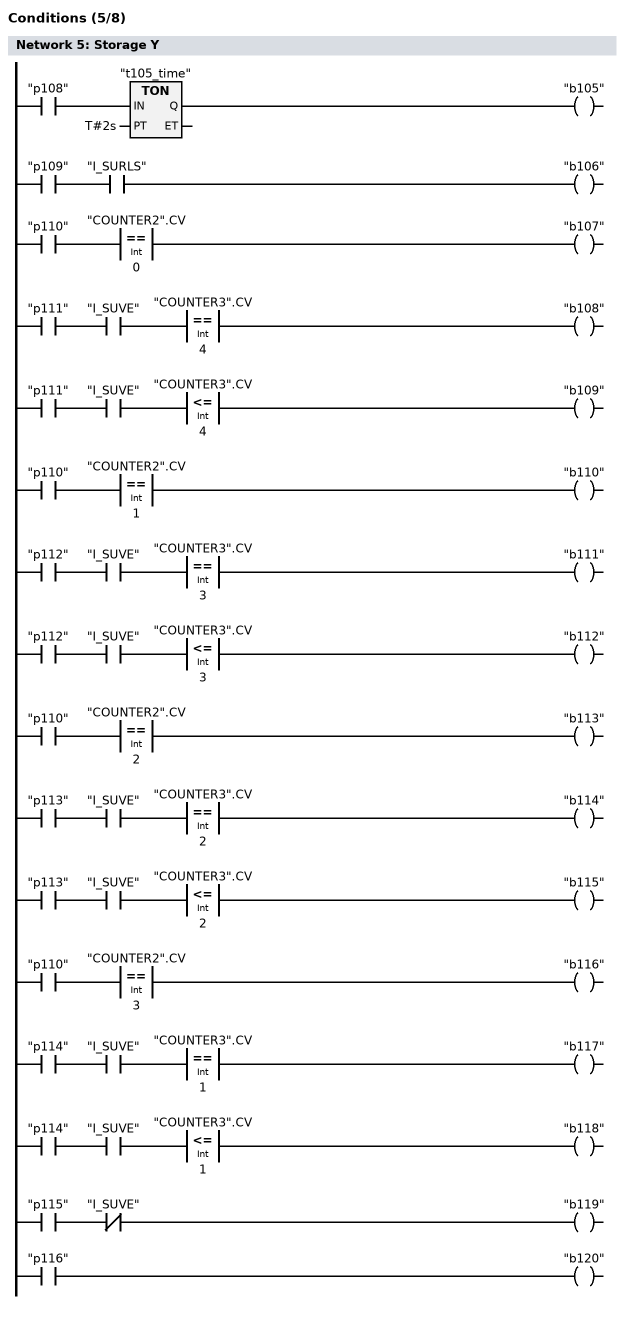
   "t105_time".TON(IN := "p108", PT := T#2s);
   "b105" := "t105_time".Q;
   "b106" := "p109" AND "I_SURLS";
   "b107" := "p110" AND ("COUNTER2".CV = 0);
   "b108" := "p111" AND "I_SUVE" AND ("COUNTER3".CV = 4);
   "b109" := "p111" AND "I_SUVE" AND ("COUNTER3".CV <= 4);
   "b110" := "p110" AND ("COUNTER2".CV = 1);
   "b111" := "p112" AND "I_SUVE" AND ("COUNTER3".CV = 3);
   "b112" := "p112" AND "I_SUVE" AND ("COUNTER3".CV <= 3);
   "b113" := "p110" AND ("COUNTER2".CV = 2);
   "b114" := "p113" AND "I_SUVE" AND ("COUNTER3".CV = 2);
   "b115" := "p113" AND "I_SUVE" AND ("COUNTER3".CV <= 2);
   "b116" := "p110" AND ("COUNTER2".CV = 3);
   "b117" := "p114" AND "I_SUVE" AND ("COUNTER3".CV = 1);
   "b118" := "p114" AND "I_SUVE" AND ("COUNTER3".CV <= 1);
   "b119" := "p115" AND NOT "I_SUVE";
   "b120" := "p116";
END_REGION

REGION Network 6: Storage X
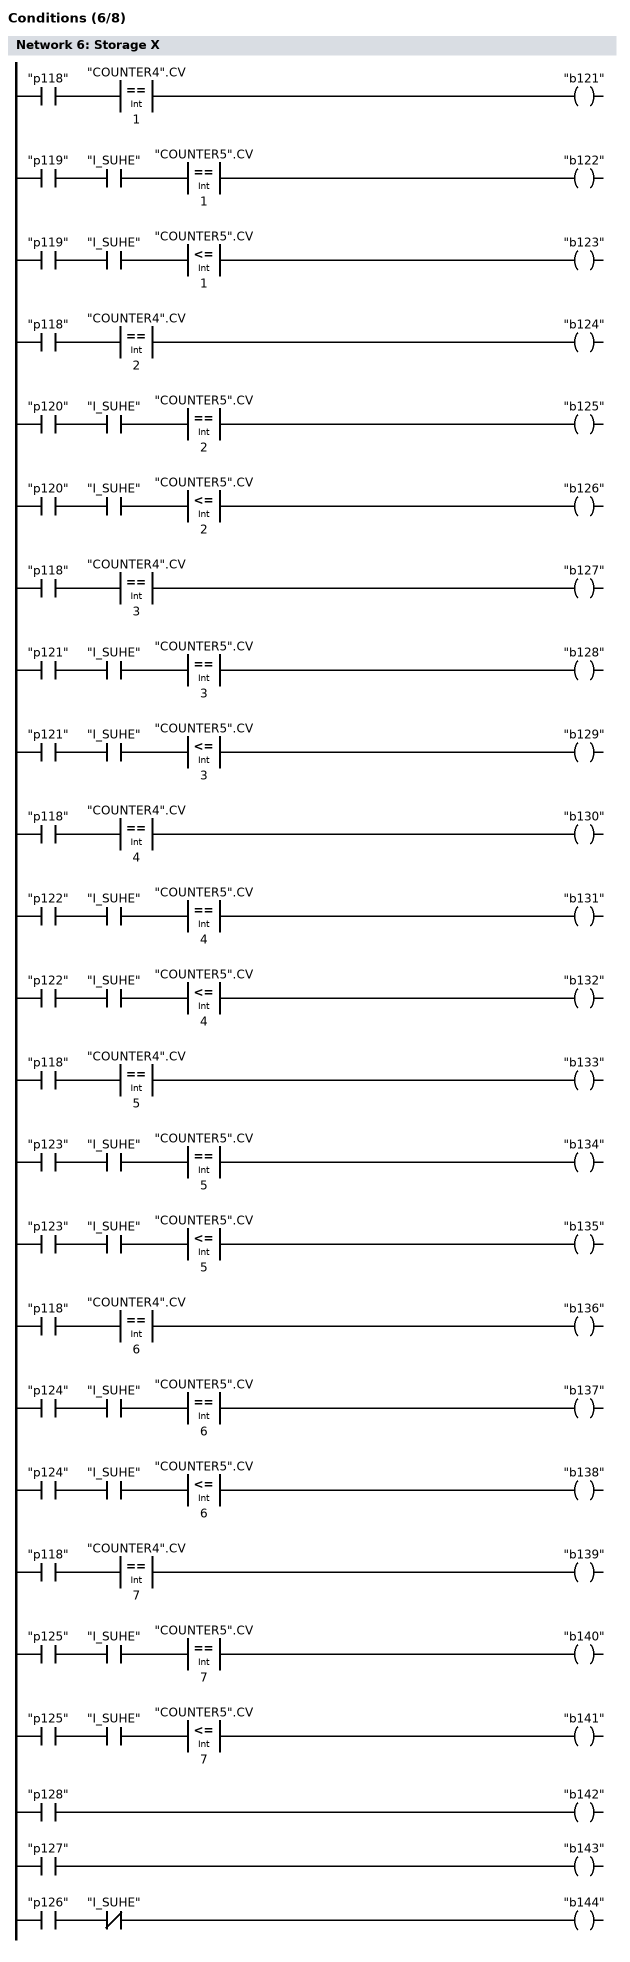
   RUNG wire#powerrail
      Contact( "p118" )
      { S7_Templates := "SrcType := Int" } EQ_Contact(in1 := "COUNTER4".CV, in2 := 1)
      Coil( "b121" )
   END_RUNG
   RUNG wire#powerrail
      Contact( "p119" )
      Contact( "I_SUHE" )
      { S7_Templates := "SrcType := Int" } EQ_Contact(in1 := "COUNTER5".CV, in2 := 1)
      Coil( "b122" )
   END_RUNG
   RUNG wire#powerrail
      Contact( "p119" )
      Contact( "I_SUHE" )
      { S7_Templates := "SrcType := Int" } LE_Contact(in1 := "COUNTER5".CV, in2 := 1)
      Coil( "b123" )
   END_RUNG
   RUNG wire#powerrail
      Contact( "p118" )
      { S7_Templates := "SrcType := Int" } EQ_Contact(in1 := "COUNTER4".CV, in2 := 2)
      Coil( "b124" )
   END_RUNG
   RUNG wire#powerrail
      Contact( "p120" )
      Contact( "I_SUHE" )
      { S7_Templates := "SrcType := Int" } EQ_Contact(in1 := "COUNTER5".CV, in2 := 2)
      Coil( "b125" )
   END_RUNG
   RUNG wire#powerrail
      Contact( "p120" )
      Contact( "I_SUHE" )
      { S7_Templates := "SrcType := Int" } LE_Contact(in1 := "COUNTER5".CV, in2 := 2)
      Coil( "b126" )
   END_RUNG
   RUNG wire#powerrail
      Contact( "p118" )
      { S7_Templates := "SrcType := Int" } EQ_Contact(in1 := "COUNTER4".CV, in2 := 3)
      Coil( "b127" )
   END_RUNG
   RUNG wire#powerrail
      Contact( "p121" )
      Contact( "I_SUHE" )
      { S7_Templates := "SrcType := Int" } EQ_Contact(in1 := "COUNTER5".CV, in2 := 3)
      Coil( "b128" )
   END_RUNG
   RUNG wire#powerrail
      Contact( "p121" )
      Contact( "I_SUHE" )
      { S7_Templates := "SrcType := Int" } LE_Contact(in1 := "COUNTER5".CV, in2 := 3)
      Coil( "b129" )
   END_RUNG
   RUNG wire#powerrail
      Contact( "p118" )
      { S7_Templates := "SrcType := Int" } EQ_Contact(in1 := "COUNTER4".CV, in2 := 4)
      Coil( "b130" )
   END_RUNG
   RUNG wire#powerrail
      Contact( "p122" )
      Contact( "I_SUHE" )
      { S7_Templates := "SrcType := Int" } EQ_Contact(in1 := "COUNTER5".CV, in2 := 4)
      Coil( "b131" )
   END_RUNG
   RUNG wire#powerrail
      Contact( "p122" )
      Contact( "I_SUHE" )
      { S7_Templates := "SrcType := Int" } LE_Contact(in1 := "COUNTER5".CV, in2 := 4)
      Coil( "b132" )
   END_RUNG
   RUNG wire#powerrail
      Contact( "p118" )
      { S7_Templates := "SrcType := Int" } EQ_Contact(in1 := "COUNTER4".CV, in2 := 5)
      Coil( "b133" )
   END_RUNG
   RUNG wire#powerrail
      Contact( "p123" )
      Contact( "I_SUHE" )
      { S7_Templates := "SrcType := Int" } EQ_Contact(in1 := "COUNTER5".CV, in2 := 5)
      Coil( "b134" )
   END_RUNG
   RUNG wire#powerrail
      Contact( "p123" )
      Contact( "I_SUHE" )
      { S7_Templates := "SrcType := Int" } LE_Contact(in1 := "COUNTER5".CV, in2 := 5)
      Coil( "b135" )
   END_RUNG
   RUNG wire#powerrail
      Contact( "p118" )
      { S7_Templates := "SrcType := Int" } EQ_Contact(in1 := "COUNTER4".CV, in2 := 6)
      Coil( "b136" )
   END_RUNG
   RUNG wire#powerrail
      Contact( "p124" )
      Contact( "I_SUHE" )
      { S7_Templates := "SrcType := Int" } EQ_Contact(in1 := "COUNTER5".CV, in2 := 6)
      Coil( "b137" )
   END_RUNG
   RUNG wire#powerrail
      Contact( "p124" )
      Contact( "I_SUHE" )
      { S7_Templates := "SrcType := Int" } LE_Contact(in1 := "COUNTER5".CV, in2 := 6)
      Coil( "b138" )
   END_RUNG
   RUNG wire#powerrail
      Contact( "p118" )
      { S7_Templates := "SrcType := Int" } EQ_Contact(in1 := "COUNTER4".CV, in2 := 7)
      Coil( "b139" )
   END_RUNG
   RUNG wire#powerrail
      Contact( "p125" )
      Contact( "I_SUHE" )
      { S7_Templates := "SrcType := Int" } EQ_Contact(in1 := "COUNTER5".CV, in2 := 7)
      Coil( "b140" )
   END_RUNG
   RUNG wire#powerrail
      Contact( "p125" )
      Contact( "I_SUHE" )
      { S7_Templates := "SrcType := Int" } LE_Contact(in1 := "COUNTER5".CV, in2 := 7)
      Coil( "b141" )
   END_RUNG
   RUNG wire#powerrail
      Contact( "p128" )
      Coil( "b142" )
   END_RUNG
   RUNG wire#powerrail
      Contact( "p127" )
      Coil( "b143" )
   END_RUNG
   RUNG wire#powerrail
      Contact( "p126" )
      I_Contact( "I_SUHE" )
      Coil( "b144" )
   END_RUNG
   // the same network as SCL:
   "b121" := "p118" AND ("COUNTER4".CV = 1);
   "b122" := "p119" AND "I_SUHE" AND ("COUNTER5".CV = 1);
   "b123" := "p119" AND "I_SUHE" AND ("COUNTER5".CV <= 1);
   "b124" := "p118" AND ("COUNTER4".CV = 2);
   "b125" := "p120" AND "I_SUHE" AND ("COUNTER5".CV = 2);
   "b126" := "p120" AND "I_SUHE" AND ("COUNTER5".CV <= 2);
   "b127" := "p118" AND ("COUNTER4".CV = 3);
   "b128" := "p121" AND "I_SUHE" AND ("COUNTER5".CV = 3);
   "b129" := "p121" AND "I_SUHE" AND ("COUNTER5".CV <= 3);
   "b130" := "p118" AND ("COUNTER4".CV = 4);
   "b131" := "p122" AND "I_SUHE" AND ("COUNTER5".CV = 4);
   "b132" := "p122" AND "I_SUHE" AND ("COUNTER5".CV <= 4);
   "b133" := "p118" AND ("COUNTER4".CV = 5);
   "b134" := "p123" AND "I_SUHE" AND ("COUNTER5".CV = 5);
   "b135" := "p123" AND "I_SUHE" AND ("COUNTER5".CV <= 5);
   "b136" := "p118" AND ("COUNTER4".CV = 6);
   "b137" := "p124" AND "I_SUHE" AND ("COUNTER5".CV = 6);
   "b138" := "p124" AND "I_SUHE" AND ("COUNTER5".CV <= 6);
   "b139" := "p118" AND ("COUNTER4".CV = 7);
   "b140" := "p125" AND "I_SUHE" AND ("COUNTER5".CV = 7);
   "b141" := "p125" AND "I_SUHE" AND ("COUNTER5".CV <= 7);
   "b142" := "p128";
   "b143" := "p127";
   "b144" := "p126" AND NOT "I_SUHE";
END_REGION

REGION Network 7: Storage piece
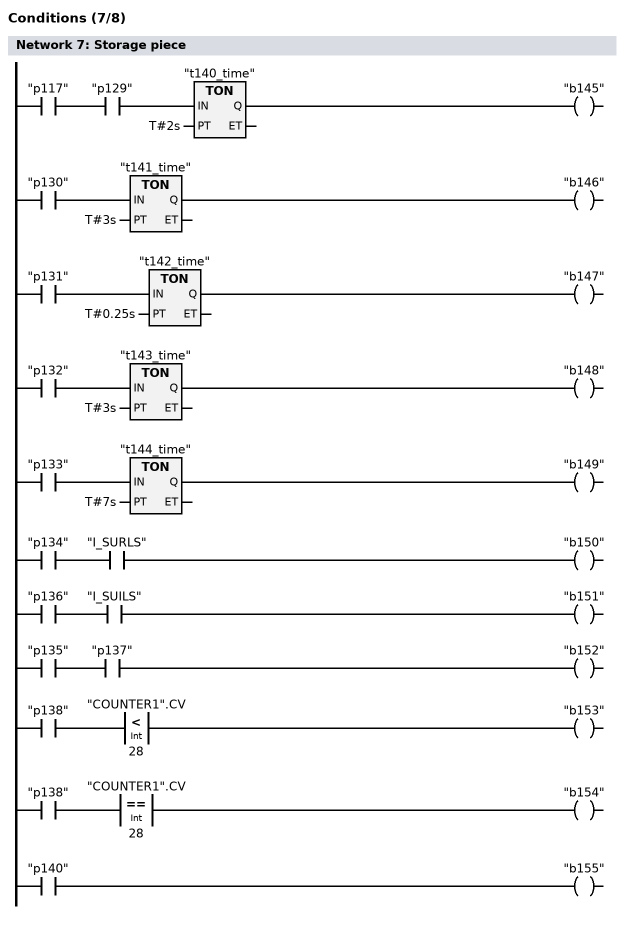
   "t140_time".TON(IN := "p117" AND "p129", PT := T#2s);
   "b145" := "t140_time".Q;
   "t141_time".TON(IN := "p130", PT := T#3s);
   "b146" := "t141_time".Q;
   "t142_time".TON(IN := "p131", PT := T#0.25s);
   "b147" := "t142_time".Q;
   "t143_time".TON(IN := "p132", PT := T#3s);
   "b148" := "t143_time".Q;
   "t144_time".TON(IN := "p133", PT := T#7s);
   "b149" := "t144_time".Q;
   "b150" := "p134" AND "I_SURLS";
   "b151" := "p136" AND "I_SUILS";
   "b152" := "p135" AND "p137";
   "b153" := "p138" AND ("COUNTER1".CV < 28);
   "b154" := "p138" AND ("COUNTER1".CV = 28);
   "b155" := "p140";
END_REGION

REGION Network 8: Arm Stop
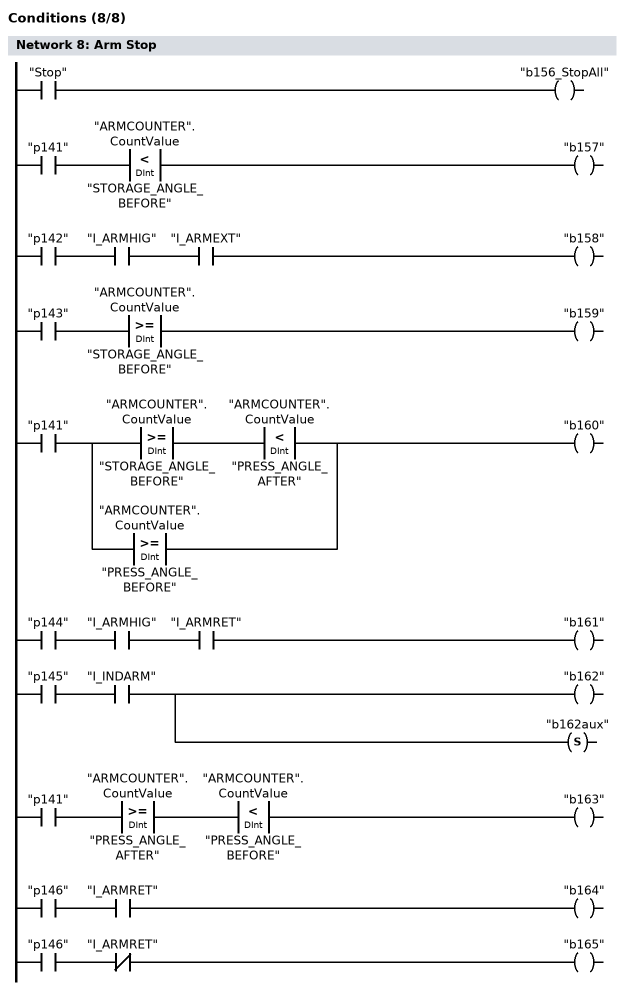
   RUNG wire#powerrail
      Contact( "Stop" )
      Coil( "b156_StopAll" )
   END_RUNG
   RUNG wire#powerrail
      Contact( "p141" )
      { S7_Templates := "SrcType := DInt" } LT_Contact(in1 := "ARMCOUNTER".CountValue, in2 := "STORAGE_ANGLE_BEFORE")
      Coil( "b157" )
   END_RUNG
   RUNG wire#powerrail
      Contact( "p142" )
      Contact( "I_ARMHIG" )
      Contact( "I_ARMEXT" )
      Coil( "b158" )
   END_RUNG
   RUNG wire#powerrail
      Contact( "p143" )
      { S7_Templates := "SrcType := DInt" } GE_Contact(in1 := "ARMCOUNTER".CountValue, in2 := "STORAGE_ANGLE_BEFORE")
      Coil( "b159" )
   END_RUNG
   RUNG wire#powerrail
      Contact( "p141" )
      wire#w1
      { S7_Templates := "SrcType := DInt" } GE_Contact(in1 := "ARMCOUNTER".CountValue, in2 := "STORAGE_ANGLE_BEFORE")
      { S7_Templates := "SrcType := DInt" } LT_Contact(in1 := "ARMCOUNTER".CountValue, in2 := "PRESS_ANGLE_AFTER")
      wire#w2
      Coil( "b160" )
   END_RUNG
   RUNG wire#w1
      { S7_Templates := "SrcType := DInt" } GE_Contact(in1 := "ARMCOUNTER".CountValue, in2 := "PRESS_ANGLE_BEFORE")
   END_RUNG wire#w2
   RUNG wire#powerrail
      Contact( "p144" )
      Contact( "I_ARMHIG" )
      Contact( "I_ARMRET" )
      Coil( "b161" )
   END_RUNG
   RUNG wire#powerrail
      Contact( "p145" )
      Contact( "I_INDARM" )
      wire#w3
      Coil( "b162" )
   END_RUNG
   RUNG wire#w3
      S_Coil( "b162aux" )
   END_RUNG
   RUNG wire#powerrail
      Contact( "p141" )
      { S7_Templates := "SrcType := DInt" } GE_Contact(in1 := "ARMCOUNTER".CountValue, in2 := "PRESS_ANGLE_AFTER")
      { S7_Templates := "SrcType := DInt" } LT_Contact(in1 := "ARMCOUNTER".CountValue, in2 := "PRESS_ANGLE_BEFORE")
      Coil( "b163" )
   END_RUNG
   RUNG wire#powerrail
      Contact( "p146" )
      Contact( "I_ARMRET" )
      Coil( "b164" )
   END_RUNG
   RUNG wire#powerrail
      Contact( "p146" )
      I_Contact( "I_ARMRET" )
      Coil( "b165" )
   END_RUNG
   // the same network as SCL:
   "b156_StopAll" := "Stop";
   "b157" := "p141" AND ("ARMCOUNTER".CountValue < "STORAGE_ANGLE_BEFORE");
   "b158" := "p142" AND "I_ARMHIG" AND "I_ARMEXT";
   "b159" := "p143" AND ("ARMCOUNTER".CountValue >= "STORAGE_ANGLE_BEFORE");
   "b160" := "p141" AND ((("ARMCOUNTER".CountValue >= "STORAGE_ANGLE_BEFORE") AND ("ARMCOUNTER".CountValue < "PRESS_ANGLE_AFTER")) OR ("ARMCOUNTER".CountValue >= "PRESS_ANGLE_BEFORE"));
   "b161" := "p144" AND "I_ARMHIG" AND "I_ARMRET";
   "b162" := "p145" AND "I_INDARM";
   IF "b162" THEN "b162aux" := TRUE; END_IF;
   "b163" := "p141" AND ("ARMCOUNTER".CountValue >= "PRESS_ANGLE_AFTER") AND ("ARMCOUNTER".CountValue < "PRESS_ANGLE_BEFORE");
   "b164" := "p146" AND "I_ARMRET";
   "b165" := "p146" AND NOT "I_ARMRET";
END_REGION
END_FUNCTION

FUNCTION "Dynamics" : Void   // FC3, LAD
{ S7_Optimized_Access := 'TRUE' }
VERSION : 0.1
BEGIN

REGION Network 1: initialization
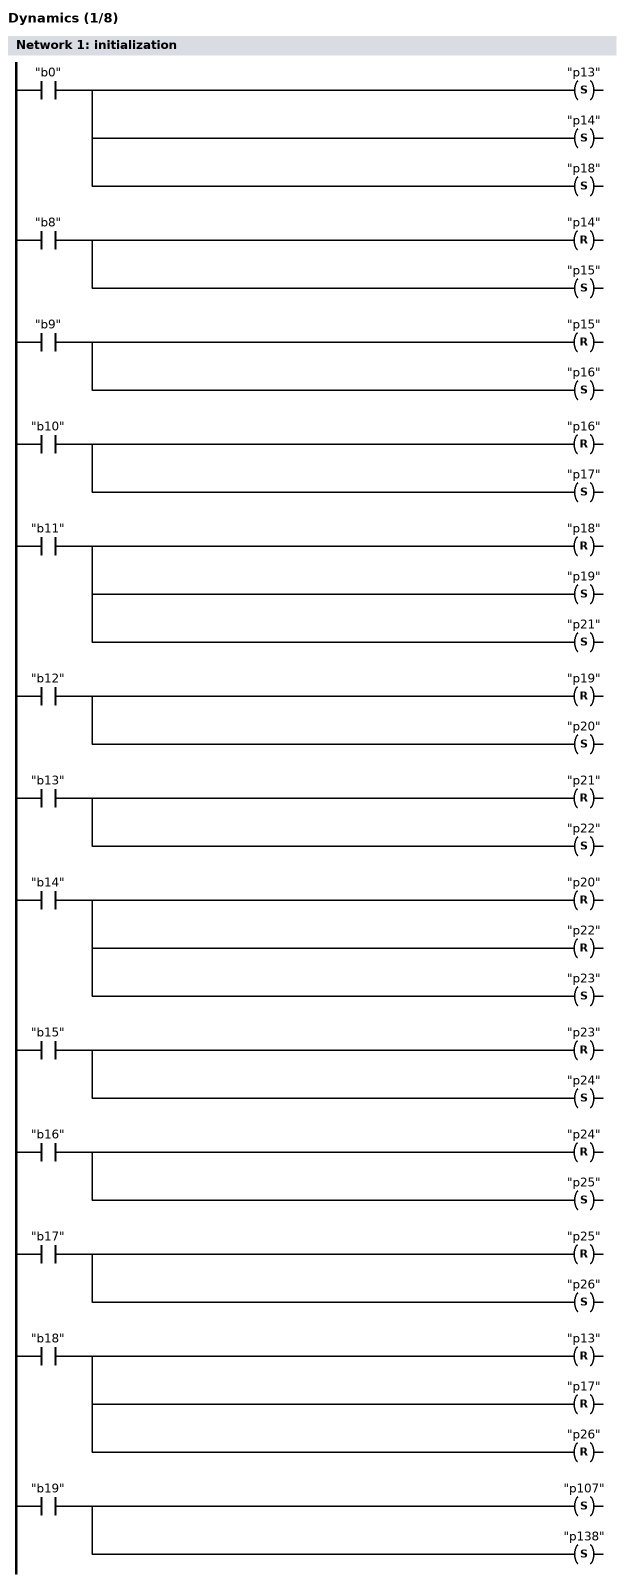
   RUNG wire#powerrail
      Contact( "b0" )
      wire#w1
      S_Coil( "p13" )
   END_RUNG
   RUNG wire#w1
      S_Coil( "p14" )
   END_RUNG
   RUNG wire#w1
      S_Coil( "p18" )
   END_RUNG
   RUNG wire#powerrail
      Contact( "b8" )
      wire#w2
      R_Coil( "p14" )
   END_RUNG
   RUNG wire#w2
      S_Coil( "p15" )
   END_RUNG
   RUNG wire#powerrail
      Contact( "b9" )
      wire#w3
      R_Coil( "p15" )
   END_RUNG
   RUNG wire#w3
      S_Coil( "p16" )
   END_RUNG
   RUNG wire#powerrail
      Contact( "b10" )
      wire#w4
      R_Coil( "p16" )
   END_RUNG
   RUNG wire#w4
      S_Coil( "p17" )
   END_RUNG
   RUNG wire#powerrail
      Contact( "b11" )
      wire#w5
      R_Coil( "p18" )
   END_RUNG
   RUNG wire#w5
      S_Coil( "p19" )
   END_RUNG
   RUNG wire#w5
      S_Coil( "p21" )
   END_RUNG
   RUNG wire#powerrail
      Contact( "b12" )
      wire#w6
      R_Coil( "p19" )
   END_RUNG
   RUNG wire#w6
      S_Coil( "p20" )
   END_RUNG
   RUNG wire#powerrail
      Contact( "b13" )
      wire#w7
      R_Coil( "p21" )
   END_RUNG
   RUNG wire#w7
      S_Coil( "p22" )
   END_RUNG
   RUNG wire#powerrail
      Contact( "b14" )
      wire#w8
      R_Coil( "p20" )
   END_RUNG
   RUNG wire#w8
      R_Coil( "p22" )
   END_RUNG
   RUNG wire#w8
      S_Coil( "p23" )
   END_RUNG
   RUNG wire#powerrail
      Contact( "b15" )
      wire#w9
      R_Coil( "p23" )
   END_RUNG
   RUNG wire#w9
      S_Coil( "p24" )
   END_RUNG
   RUNG wire#powerrail
      Contact( "b16" )
      wire#w10
      R_Coil( "p24" )
   END_RUNG
   RUNG wire#w10
      S_Coil( "p25" )
   END_RUNG
   RUNG wire#powerrail
      Contact( "b17" )
      wire#w11
      R_Coil( "p25" )
   END_RUNG
   RUNG wire#w11
      S_Coil( "p26" )
   END_RUNG
   RUNG wire#powerrail
      Contact( "b18" )
      wire#w12
      R_Coil( "p13" )
   END_RUNG
   RUNG wire#w12
      R_Coil( "p17" )
   END_RUNG
   RUNG wire#w12
      R_Coil( "p26" )
   END_RUNG
   RUNG wire#powerrail
      Contact( "b19" )
      wire#w13
      S_Coil( "p107" )
   END_RUNG
   RUNG wire#w13
      S_Coil( "p138" )
   END_RUNG
   // the same network as SCL:
   IF "b0" THEN
       "p13" := TRUE;
       "p14" := TRUE;
       "p18" := TRUE;
   END_IF;
   IF "b8" THEN
       "p14" := FALSE;
       "p15" := TRUE;
   END_IF;
   IF "b9" THEN
       "p15" := FALSE;
       "p16" := TRUE;
   END_IF;
   IF "b10" THEN
       "p16" := FALSE;
       "p17" := TRUE;
   END_IF;
   IF "b11" THEN
       "p18" := FALSE;
       "p19" := TRUE;
       "p21" := TRUE;
   END_IF;
   IF "b12" THEN
       "p19" := FALSE;
       "p20" := TRUE;
   END_IF;
   IF "b13" THEN
       "p21" := FALSE;
       "p22" := TRUE;
   END_IF;
   IF "b14" THEN
       "p20" := FALSE;
       "p22" := FALSE;
       "p23" := TRUE;
   END_IF;
   IF "b15" THEN
       "p23" := FALSE;
       "p24" := TRUE;
   END_IF;
   IF "b16" THEN
       "p24" := FALSE;
       "p25" := TRUE;
   END_IF;
   IF "b17" THEN
       "p25" := FALSE;
       "p26" := TRUE;
   END_IF;
   IF "b18" THEN
       "p13" := FALSE;
       "p17" := FALSE;
       "p26" := FALSE;
   END_IF;
   IF "b19" THEN
       "p107" := TRUE;
       "p138" := TRUE;
   END_IF;
END_REGION

REGION Network 3: Arm Belt to Press
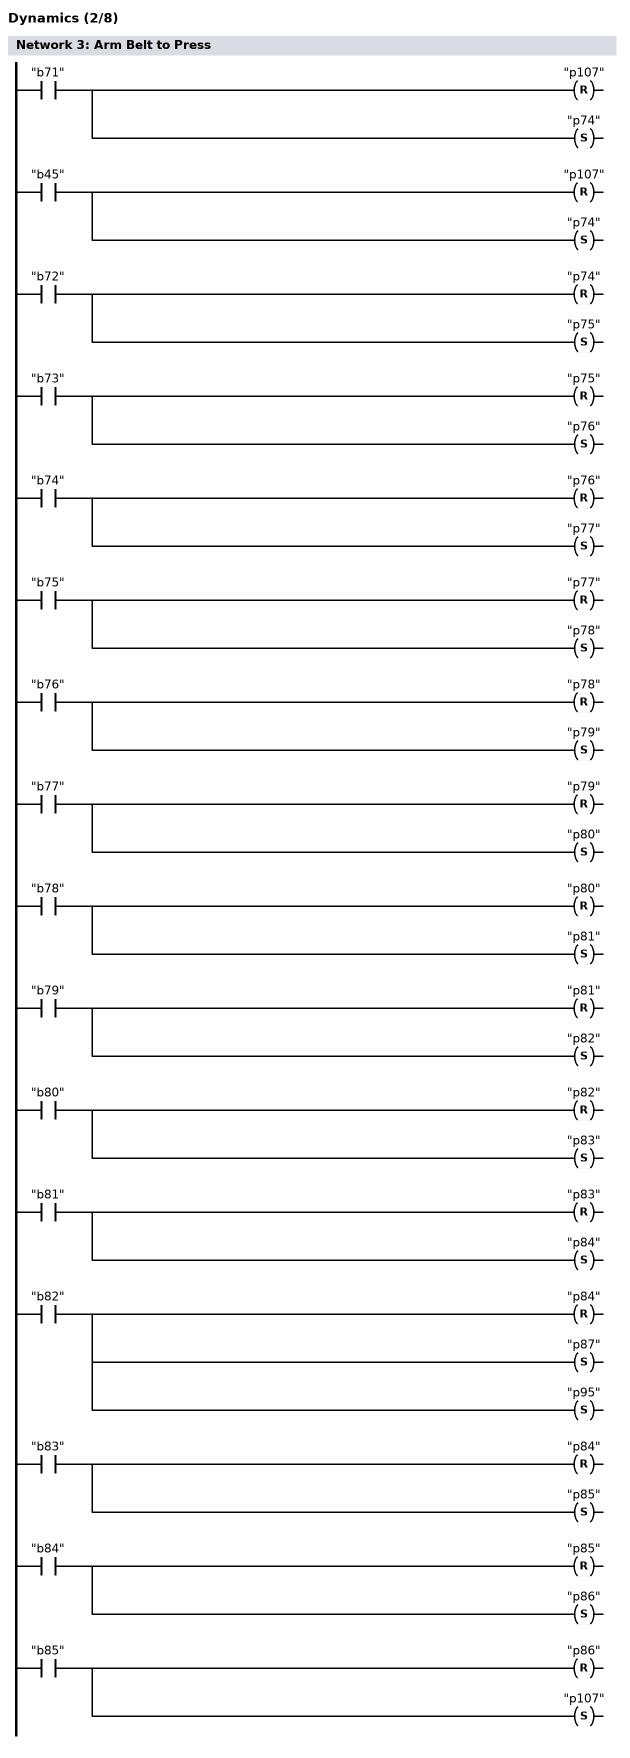
   RUNG wire#powerrail
      Contact( "b71" )
      wire#w1
      R_Coil( "p107" )
   END_RUNG
   RUNG wire#w1
      S_Coil( "p74" )
   END_RUNG
   RUNG wire#powerrail
      Contact( "b45" )
      wire#w2
      R_Coil( "p107" )
   END_RUNG
   RUNG wire#w2
      S_Coil( "p74" )
   END_RUNG
   RUNG wire#powerrail
      Contact( "b72" )
      wire#w3
      R_Coil( "p74" )
   END_RUNG
   RUNG wire#w3
      S_Coil( "p75" )
   END_RUNG
   RUNG wire#powerrail
      Contact( "b73" )
      wire#w4
      R_Coil( "p75" )
   END_RUNG
   RUNG wire#w4
      S_Coil( "p76" )
   END_RUNG
   RUNG wire#powerrail
      Contact( "b74" )
      wire#w5
      R_Coil( "p76" )
   END_RUNG
   RUNG wire#w5
      S_Coil( "p77" )
   END_RUNG
   RUNG wire#powerrail
      Contact( "b75" )
      wire#w6
      R_Coil( "p77" )
   END_RUNG
   RUNG wire#w6
      S_Coil( "p78" )
   END_RUNG
   RUNG wire#powerrail
      Contact( "b76" )
      wire#w7
      R_Coil( "p78" )
   END_RUNG
   RUNG wire#w7
      S_Coil( "p79" )
   END_RUNG
   RUNG wire#powerrail
      Contact( "b77" )
      wire#w8
      R_Coil( "p79" )
   END_RUNG
   RUNG wire#w8
      S_Coil( "p80" )
   END_RUNG
   RUNG wire#powerrail
      Contact( "b78" )
      wire#w9
      R_Coil( "p80" )
   END_RUNG
   RUNG wire#w9
      S_Coil( "p81" )
   END_RUNG
   RUNG wire#powerrail
      Contact( "b79" )
      wire#w10
      R_Coil( "p81" )
   END_RUNG
   RUNG wire#w10
      S_Coil( "p82" )
   END_RUNG
   RUNG wire#powerrail
      Contact( "b80" )
      wire#w11
      R_Coil( "p82" )
   END_RUNG
   RUNG wire#w11
      S_Coil( "p83" )
   END_RUNG
   RUNG wire#powerrail
      Contact( "b81" )
      wire#w12
      R_Coil( "p83" )
   END_RUNG
   RUNG wire#w12
      S_Coil( "p84" )
   END_RUNG
   RUNG wire#powerrail
      Contact( "b82" )
      wire#w13
      R_Coil( "p84" )
   END_RUNG
   RUNG wire#w13
      S_Coil( "p87" )
   END_RUNG
   RUNG wire#w13
      S_Coil( "p95" )
   END_RUNG
   RUNG wire#powerrail
      Contact( "b83" )
      wire#w14
      R_Coil( "p84" )
   END_RUNG
   RUNG wire#w14
      S_Coil( "p85" )
   END_RUNG
   RUNG wire#powerrail
      Contact( "b84" )
      wire#w15
      R_Coil( "p85" )
   END_RUNG
   RUNG wire#w15
      S_Coil( "p86" )
   END_RUNG
   RUNG wire#powerrail
      Contact( "b85" )
      wire#w16
      R_Coil( "p86" )
   END_RUNG
   RUNG wire#w16
      S_Coil( "p107" )
   END_RUNG
   // the same network as SCL:
   IF "b71" THEN
       "p107" := FALSE;
       "p74" := TRUE;
   END_IF;
   IF "b45" THEN
       "p107" := FALSE;
       "p74" := TRUE;
   END_IF;
   IF "b72" THEN
       "p74" := FALSE;
       "p75" := TRUE;
   END_IF;
   IF "b73" THEN
       "p75" := FALSE;
       "p76" := TRUE;
   END_IF;
   IF "b74" THEN
       "p76" := FALSE;
       "p77" := TRUE;
   END_IF;
   IF "b75" THEN
       "p77" := FALSE;
       "p78" := TRUE;
   END_IF;
   IF "b76" THEN
       "p78" := FALSE;
       "p79" := TRUE;
   END_IF;
   IF "b77" THEN
       "p79" := FALSE;
       "p80" := TRUE;
   END_IF;
   IF "b78" THEN
       "p80" := FALSE;
       "p81" := TRUE;
   END_IF;
   IF "b79" THEN
       "p81" := FALSE;
       "p82" := TRUE;
   END_IF;
   IF "b80" THEN
       "p82" := FALSE;
       "p83" := TRUE;
   END_IF;
   IF "b81" THEN
       "p83" := FALSE;
       "p84" := TRUE;
   END_IF;
   IF "b82" THEN
       "p84" := FALSE;
       "p87" := TRUE;
       "p95" := TRUE;
   END_IF;
   IF "b83" THEN
       "p84" := FALSE;
       "p85" := TRUE;
   END_IF;
   IF "b84" THEN
       "p85" := FALSE;
       "p86" := TRUE;
   END_IF;
   IF "b85" THEN
       "p86" := FALSE;
       "p107" := TRUE;
   END_IF;
END_REGION

REGION Network 4: Assembly Unit
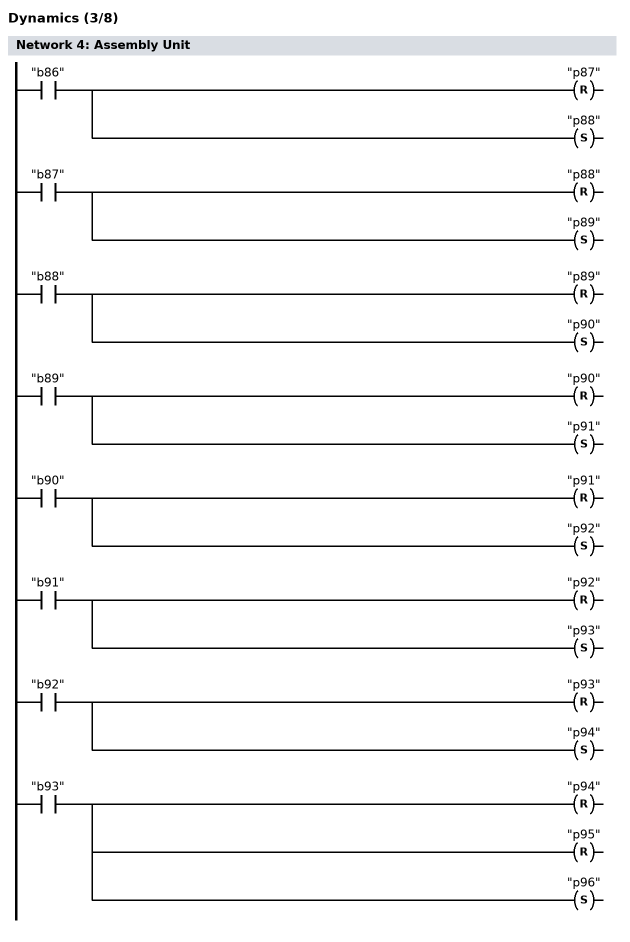
   RUNG wire#powerrail
      Contact( "b86" )
      wire#w1
      R_Coil( "p87" )
   END_RUNG
   RUNG wire#w1
      S_Coil( "p88" )
   END_RUNG
   RUNG wire#powerrail
      Contact( "b87" )
      wire#w2
      R_Coil( "p88" )
   END_RUNG
   RUNG wire#w2
      S_Coil( "p89" )
   END_RUNG
   RUNG wire#powerrail
      Contact( "b88" )
      wire#w3
      R_Coil( "p89" )
   END_RUNG
   RUNG wire#w3
      S_Coil( "p90" )
   END_RUNG
   RUNG wire#powerrail
      Contact( "b89" )
      wire#w4
      R_Coil( "p90" )
   END_RUNG
   RUNG wire#w4
      S_Coil( "p91" )
   END_RUNG
   RUNG wire#powerrail
      Contact( "b90" )
      wire#w5
      R_Coil( "p91" )
   END_RUNG
   RUNG wire#w5
      S_Coil( "p92" )
   END_RUNG
   RUNG wire#powerrail
      Contact( "b91" )
      wire#w6
      R_Coil( "p92" )
   END_RUNG
   RUNG wire#w6
      S_Coil( "p93" )
   END_RUNG
   RUNG wire#powerrail
      Contact( "b92" )
      wire#w7
      R_Coil( "p93" )
   END_RUNG
   RUNG wire#w7
      S_Coil( "p94" )
   END_RUNG
   RUNG wire#powerrail
      Contact( "b93" )
      wire#w8
      R_Coil( "p94" )
   END_RUNG
   RUNG wire#w8
      R_Coil( "p95" )
   END_RUNG
   RUNG wire#w8
      S_Coil( "p96" )
   END_RUNG
   // the same network as SCL:
   IF "b86" THEN
       "p87" := FALSE;
       "p88" := TRUE;
   END_IF;
   IF "b87" THEN
       "p88" := FALSE;
       "p89" := TRUE;
   END_IF;
   IF "b88" THEN
       "p89" := FALSE;
       "p90" := TRUE;
   END_IF;
   IF "b89" THEN
       "p90" := FALSE;
       "p91" := TRUE;
   END_IF;
   IF "b90" THEN
       "p91" := FALSE;
       "p92" := TRUE;
   END_IF;
   IF "b91" THEN
       "p92" := FALSE;
       "p93" := TRUE;
   END_IF;
   IF "b92" THEN
       "p93" := FALSE;
       "p94" := TRUE;
   END_IF;
   IF "b93" THEN
       "p94" := FALSE;
       "p95" := FALSE;
       "p96" := TRUE;
   END_IF;
END_REGION

REGION Network 5: Arm Press To Storage Unit
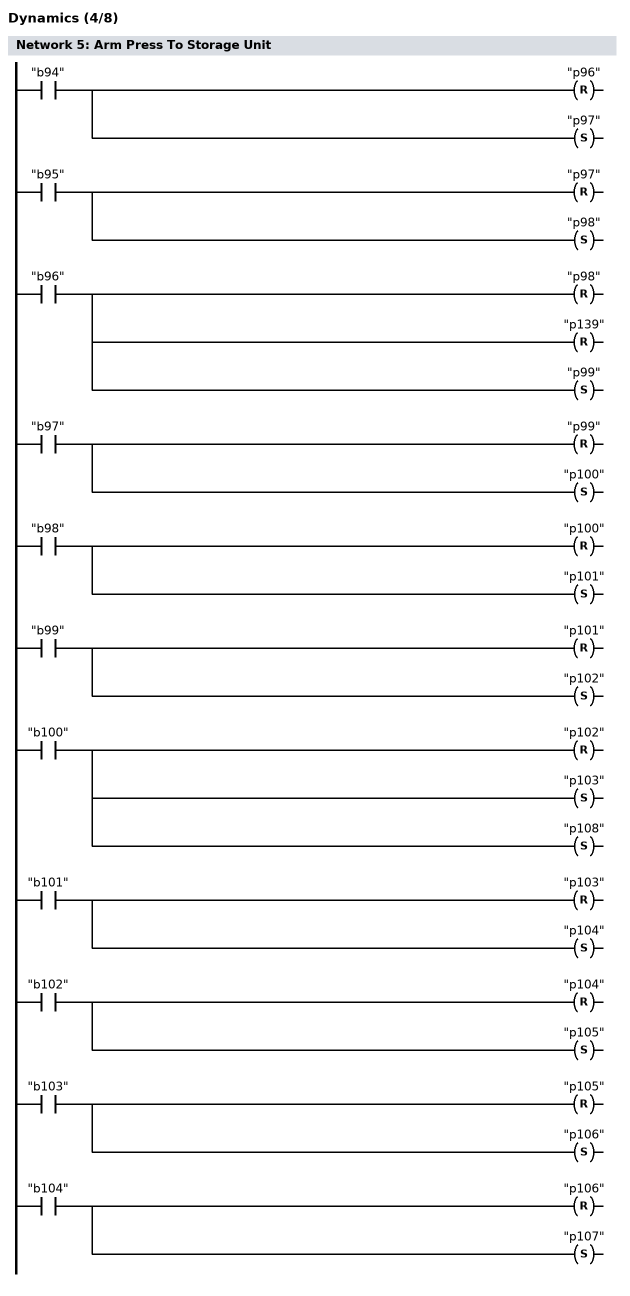
   RUNG wire#powerrail
      Contact( "b94" )
      wire#w1
      R_Coil( "p96" )
   END_RUNG
   RUNG wire#w1
      S_Coil( "p97" )
   END_RUNG
   RUNG wire#powerrail
      Contact( "b95" )
      wire#w2
      R_Coil( "p97" )
   END_RUNG
   RUNG wire#w2
      S_Coil( "p98" )
   END_RUNG
   RUNG wire#powerrail
      Contact( "b96" )
      wire#w3
      R_Coil( "p98" )
   END_RUNG
   RUNG wire#w3
      R_Coil( "p139" )
   END_RUNG
   RUNG wire#w3
      S_Coil( "p99" )
   END_RUNG
   RUNG wire#powerrail
      Contact( "b97" )
      wire#w4
      R_Coil( "p99" )
   END_RUNG
   RUNG wire#w4
      S_Coil( "p100" )
   END_RUNG
   RUNG wire#powerrail
      Contact( "b98" )
      wire#w5
      R_Coil( "p100" )
   END_RUNG
   RUNG wire#w5
      S_Coil( "p101" )
   END_RUNG
   RUNG wire#powerrail
      Contact( "b99" )
      wire#w6
      R_Coil( "p101" )
   END_RUNG
   RUNG wire#w6
      S_Coil( "p102" )
   END_RUNG
   RUNG wire#powerrail
      Contact( "b100" )
      wire#w7
      R_Coil( "p102" )
   END_RUNG
   RUNG wire#w7
      S_Coil( "p103" )
   END_RUNG
   RUNG wire#w7
      S_Coil( "p108" )
   END_RUNG
   RUNG wire#powerrail
      Contact( "b101" )
      wire#w8
      R_Coil( "p103" )
   END_RUNG
   RUNG wire#w8
      S_Coil( "p104" )
   END_RUNG
   RUNG wire#powerrail
      Contact( "b102" )
      wire#w9
      R_Coil( "p104" )
   END_RUNG
   RUNG wire#w9
      S_Coil( "p105" )
   END_RUNG
   RUNG wire#powerrail
      Contact( "b103" )
      wire#w10
      R_Coil( "p105" )
   END_RUNG
   RUNG wire#w10
      S_Coil( "p106" )
   END_RUNG
   RUNG wire#powerrail
      Contact( "b104" )
      wire#w11
      R_Coil( "p106" )
   END_RUNG
   RUNG wire#w11
      S_Coil( "p107" )
   END_RUNG
   // the same network as SCL:
   IF "b94" THEN
       "p96" := FALSE;
       "p97" := TRUE;
   END_IF;
   IF "b95" THEN
       "p97" := FALSE;
       "p98" := TRUE;
   END_IF;
   IF "b96" THEN
       "p98" := FALSE;
       "p139" := FALSE;
       "p99" := TRUE;
   END_IF;
   IF "b97" THEN
       "p99" := FALSE;
       "p100" := TRUE;
   END_IF;
   IF "b98" THEN
       "p100" := FALSE;
       "p101" := TRUE;
   END_IF;
   IF "b99" THEN
       "p101" := FALSE;
       "p102" := TRUE;
   END_IF;
   IF "b100" THEN
       "p102" := FALSE;
       "p103" := TRUE;
       "p108" := TRUE;
   END_IF;
   IF "b101" THEN
       "p103" := FALSE;
       "p104" := TRUE;
   END_IF;
   IF "b102" THEN
       "p104" := FALSE;
       "p105" := TRUE;
   END_IF;
   IF "b103" THEN
       "p105" := FALSE;
       "p106" := TRUE;
   END_IF;
   IF "b104" THEN
       "p106" := FALSE;
       "p107" := TRUE;
   END_IF;
END_REGION

REGION Network 6: Storage Y
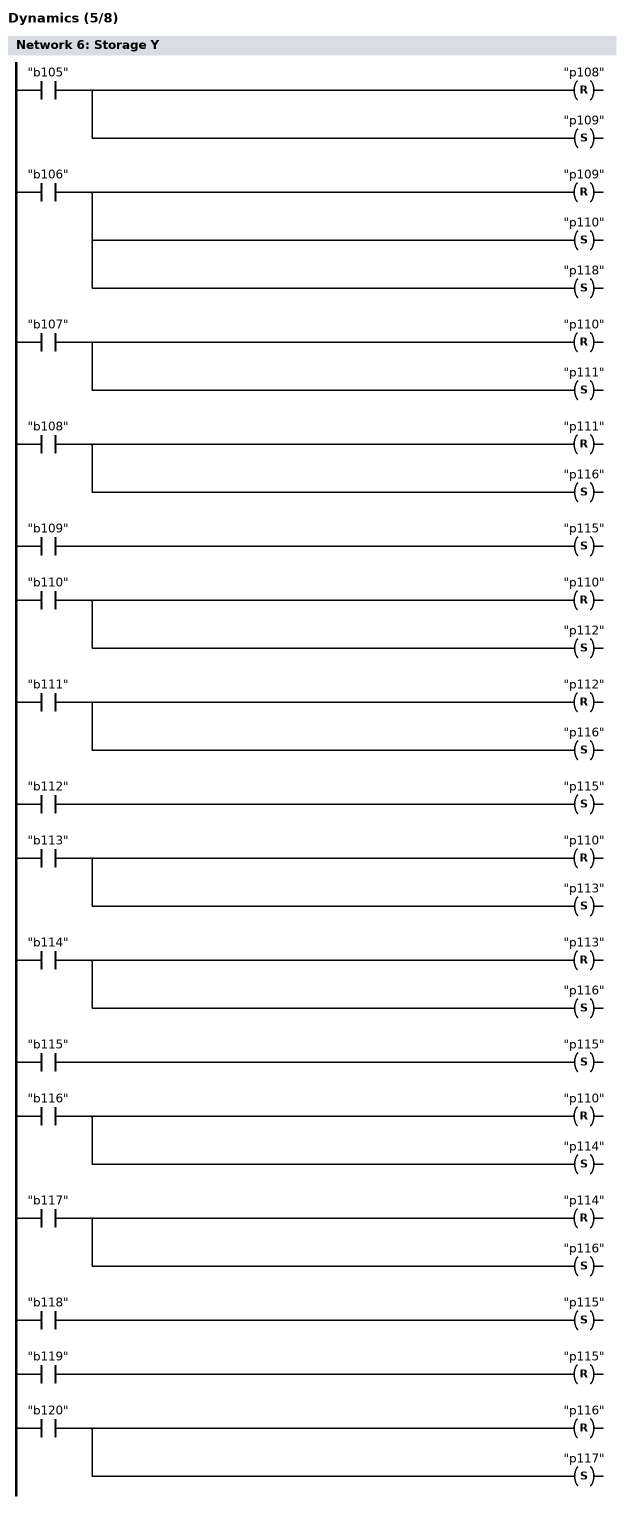
   RUNG wire#powerrail
      Contact( "b105" )
      wire#w1
      R_Coil( "p108" )
   END_RUNG
   RUNG wire#w1
      S_Coil( "p109" )
   END_RUNG
   RUNG wire#powerrail
      Contact( "b106" )
      wire#w2
      R_Coil( "p109" )
   END_RUNG
   RUNG wire#w2
      S_Coil( "p110" )
   END_RUNG
   RUNG wire#w2
      S_Coil( "p118" )
   END_RUNG
   RUNG wire#powerrail
      Contact( "b107" )
      wire#w3
      R_Coil( "p110" )
   END_RUNG
   RUNG wire#w3
      S_Coil( "p111" )
   END_RUNG
   RUNG wire#powerrail
      Contact( "b108" )
      wire#w4
      R_Coil( "p111" )
   END_RUNG
   RUNG wire#w4
      S_Coil( "p116" )
   END_RUNG
   RUNG wire#powerrail
      Contact( "b109" )
      S_Coil( "p115" )
   END_RUNG
   RUNG wire#powerrail
      Contact( "b110" )
      wire#w5
      R_Coil( "p110" )
   END_RUNG
   RUNG wire#w5
      S_Coil( "p112" )
   END_RUNG
   RUNG wire#powerrail
      Contact( "b111" )
      wire#w6
      R_Coil( "p112" )
   END_RUNG
   RUNG wire#w6
      S_Coil( "p116" )
   END_RUNG
   RUNG wire#powerrail
      Contact( "b112" )
      S_Coil( "p115" )
   END_RUNG
   RUNG wire#powerrail
      Contact( "b113" )
      wire#w7
      R_Coil( "p110" )
   END_RUNG
   RUNG wire#w7
      S_Coil( "p113" )
   END_RUNG
   RUNG wire#powerrail
      Contact( "b114" )
      wire#w8
      R_Coil( "p113" )
   END_RUNG
   RUNG wire#w8
      S_Coil( "p116" )
   END_RUNG
   RUNG wire#powerrail
      Contact( "b115" )
      S_Coil( "p115" )
   END_RUNG
   RUNG wire#powerrail
      Contact( "b116" )
      wire#w9
      R_Coil( "p110" )
   END_RUNG
   RUNG wire#w9
      S_Coil( "p114" )
   END_RUNG
   RUNG wire#powerrail
      Contact( "b117" )
      wire#w10
      R_Coil( "p114" )
   END_RUNG
   RUNG wire#w10
      S_Coil( "p116" )
   END_RUNG
   RUNG wire#powerrail
      Contact( "b118" )
      S_Coil( "p115" )
   END_RUNG
   RUNG wire#powerrail
      Contact( "b119" )
      R_Coil( "p115" )
   END_RUNG
   RUNG wire#powerrail
      Contact( "b120" )
      wire#w11
      R_Coil( "p116" )
   END_RUNG
   RUNG wire#w11
      S_Coil( "p117" )
   END_RUNG
   // the same network as SCL:
   IF "b105" THEN
       "p108" := FALSE;
       "p109" := TRUE;
   END_IF;
   IF "b106" THEN
       "p109" := FALSE;
       "p110" := TRUE;
       "p118" := TRUE;
   END_IF;
   IF "b107" THEN
       "p110" := FALSE;
       "p111" := TRUE;
   END_IF;
   IF "b108" THEN
       "p111" := FALSE;
       "p116" := TRUE;
   END_IF;
   IF "b109" THEN "p115" := TRUE; END_IF;
   IF "b110" THEN
       "p110" := FALSE;
       "p112" := TRUE;
   END_IF;
   IF "b111" THEN
       "p112" := FALSE;
       "p116" := TRUE;
   END_IF;
   IF "b112" THEN "p115" := TRUE; END_IF;
   IF "b113" THEN
       "p110" := FALSE;
       "p113" := TRUE;
   END_IF;
   IF "b114" THEN
       "p113" := FALSE;
       "p116" := TRUE;
   END_IF;
   IF "b115" THEN "p115" := TRUE; END_IF;
   IF "b116" THEN
       "p110" := FALSE;
       "p114" := TRUE;
   END_IF;
   IF "b117" THEN
       "p114" := FALSE;
       "p116" := TRUE;
   END_IF;
   IF "b118" THEN "p115" := TRUE; END_IF;
   IF "b119" THEN "p115" := FALSE; END_IF;
   IF "b120" THEN
       "p116" := FALSE;
       "p117" := TRUE;
   END_IF;
END_REGION

REGION Network 7: Storage X
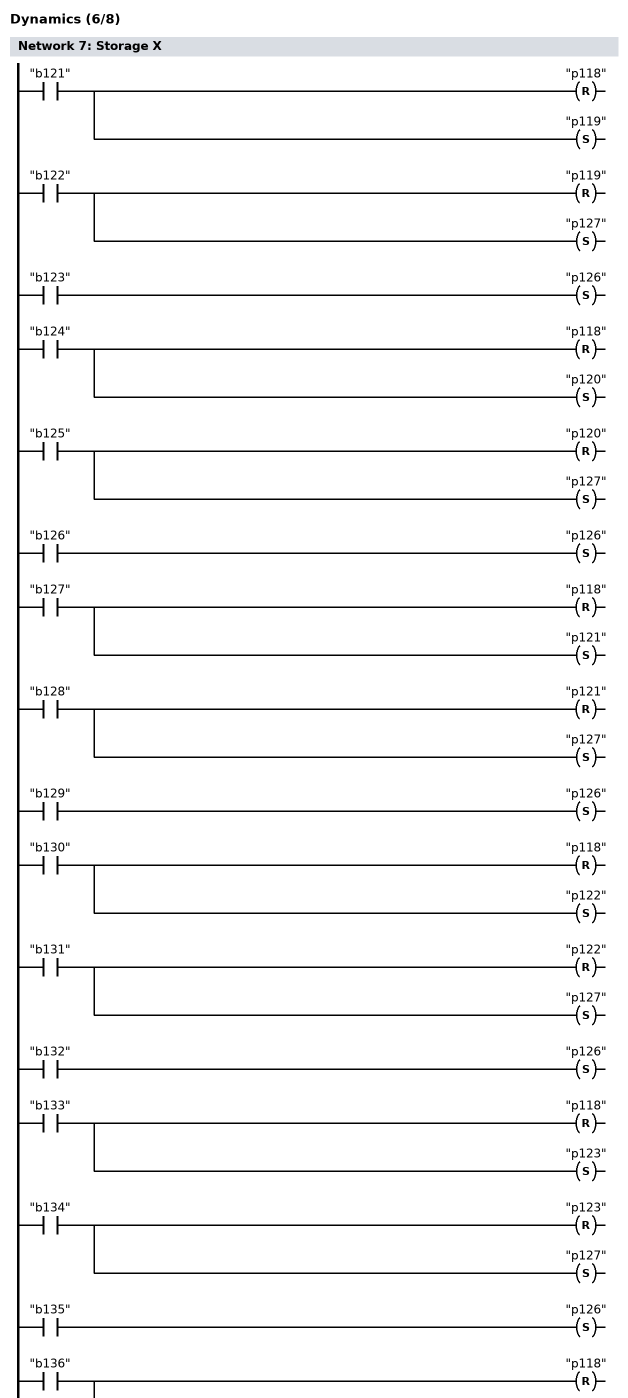
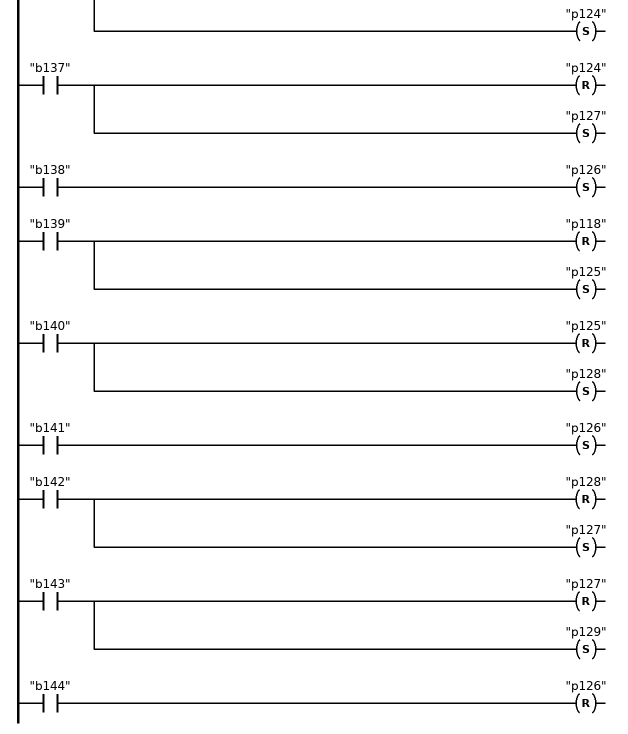
   RUNG wire#powerrail
      Contact( "b121" )
      wire#w1
      R_Coil( "p118" )
   END_RUNG
   RUNG wire#w1
      S_Coil( "p119" )
   END_RUNG
   RUNG wire#powerrail
      Contact( "b122" )
      wire#w2
      R_Coil( "p119" )
   END_RUNG
   RUNG wire#w2
      S_Coil( "p127" )
   END_RUNG
   RUNG wire#powerrail
      Contact( "b123" )
      S_Coil( "p126" )
   END_RUNG
   RUNG wire#powerrail
      Contact( "b124" )
      wire#w3
      R_Coil( "p118" )
   END_RUNG
   RUNG wire#w3
      S_Coil( "p120" )
   END_RUNG
   RUNG wire#powerrail
      Contact( "b125" )
      wire#w4
      R_Coil( "p120" )
   END_RUNG
   RUNG wire#w4
      S_Coil( "p127" )
   END_RUNG
   RUNG wire#powerrail
      Contact( "b126" )
      S_Coil( "p126" )
   END_RUNG
   RUNG wire#powerrail
      Contact( "b127" )
      wire#w5
      R_Coil( "p118" )
   END_RUNG
   RUNG wire#w5
      S_Coil( "p121" )
   END_RUNG
   RUNG wire#powerrail
      Contact( "b128" )
      wire#w6
      R_Coil( "p121" )
   END_RUNG
   RUNG wire#w6
      S_Coil( "p127" )
   END_RUNG
   RUNG wire#powerrail
      Contact( "b129" )
      S_Coil( "p126" )
   END_RUNG
   RUNG wire#powerrail
      Contact( "b130" )
      wire#w7
      R_Coil( "p118" )
   END_RUNG
   RUNG wire#w7
      S_Coil( "p122" )
   END_RUNG
   RUNG wire#powerrail
      Contact( "b131" )
      wire#w8
      R_Coil( "p122" )
   END_RUNG
   RUNG wire#w8
      S_Coil( "p127" )
   END_RUNG
   RUNG wire#powerrail
      Contact( "b132" )
      S_Coil( "p126" )
   END_RUNG
   RUNG wire#powerrail
      Contact( "b133" )
      wire#w9
      R_Coil( "p118" )
   END_RUNG
   RUNG wire#w9
      S_Coil( "p123" )
   END_RUNG
   RUNG wire#powerrail
      Contact( "b134" )
      wire#w10
      R_Coil( "p123" )
   END_RUNG
   RUNG wire#w10
      S_Coil( "p127" )
   END_RUNG
   RUNG wire#powerrail
      Contact( "b135" )
      S_Coil( "p126" )
   END_RUNG
   RUNG wire#powerrail
      Contact( "b136" )
      wire#w11
      R_Coil( "p118" )
   END_RUNG
   RUNG wire#w11
      S_Coil( "p124" )
   END_RUNG
   RUNG wire#powerrail
      Contact( "b137" )
      wire#w12
      R_Coil( "p124" )
   END_RUNG
   RUNG wire#w12
      S_Coil( "p127" )
   END_RUNG
   RUNG wire#powerrail
      Contact( "b138" )
      S_Coil( "p126" )
   END_RUNG
   RUNG wire#powerrail
      Contact( "b139" )
      wire#w13
      R_Coil( "p118" )
   END_RUNG
   RUNG wire#w13
      S_Coil( "p125" )
   END_RUNG
   RUNG wire#powerrail
      Contact( "b140" )
      wire#w14
      R_Coil( "p125" )
   END_RUNG
   RUNG wire#w14
      S_Coil( "p128" )
   END_RUNG
   RUNG wire#powerrail
      Contact( "b141" )
      S_Coil( "p126" )
   END_RUNG
   RUNG wire#powerrail
      Contact( "b142" )
      wire#w15
      R_Coil( "p128" )
   END_RUNG
   RUNG wire#w15
      S_Coil( "p127" )
   END_RUNG
   RUNG wire#powerrail
      Contact( "b143" )
      wire#w16
      R_Coil( "p127" )
   END_RUNG
   RUNG wire#w16
      S_Coil( "p129" )
   END_RUNG
   RUNG wire#powerrail
      Contact( "b144" )
      R_Coil( "p126" )
   END_RUNG
   // the same network as SCL:
   IF "b121" THEN
       "p118" := FALSE;
       "p119" := TRUE;
   END_IF;
   IF "b122" THEN
       "p119" := FALSE;
       "p127" := TRUE;
   END_IF;
   IF "b123" THEN "p126" := TRUE; END_IF;
   IF "b124" THEN
       "p118" := FALSE;
       "p120" := TRUE;
   END_IF;
   IF "b125" THEN
       "p120" := FALSE;
       "p127" := TRUE;
   END_IF;
   IF "b126" THEN "p126" := TRUE; END_IF;
   IF "b127" THEN
       "p118" := FALSE;
       "p121" := TRUE;
   END_IF;
   IF "b128" THEN
       "p121" := FALSE;
       "p127" := TRUE;
   END_IF;
   IF "b129" THEN "p126" := TRUE; END_IF;
   IF "b130" THEN
       "p118" := FALSE;
       "p122" := TRUE;
   END_IF;
   IF "b131" THEN
       "p122" := FALSE;
       "p127" := TRUE;
   END_IF;
   IF "b132" THEN "p126" := TRUE; END_IF;
   IF "b133" THEN
       "p118" := FALSE;
       "p123" := TRUE;
   END_IF;
   IF "b134" THEN
       "p123" := FALSE;
       "p127" := TRUE;
   END_IF;
   IF "b135" THEN "p126" := TRUE; END_IF;
   IF "b136" THEN
       "p118" := FALSE;
       "p124" := TRUE;
   END_IF;
   IF "b137" THEN
       "p124" := FALSE;
       "p127" := TRUE;
   END_IF;
   IF "b138" THEN "p126" := TRUE; END_IF;
   IF "b139" THEN
       "p118" := FALSE;
       "p125" := TRUE;
   END_IF;
   IF "b140" THEN
       "p125" := FALSE;
       "p128" := TRUE;
   END_IF;
   IF "b141" THEN "p126" := TRUE; END_IF;
   IF "b142" THEN
       "p128" := FALSE;
       "p127" := TRUE;
   END_IF;
   IF "b143" THEN
       "p127" := FALSE;
       "p129" := TRUE;
   END_IF;
   IF "b144" THEN "p126" := FALSE; END_IF;
END_REGION

REGION Network 8: Storage Piece
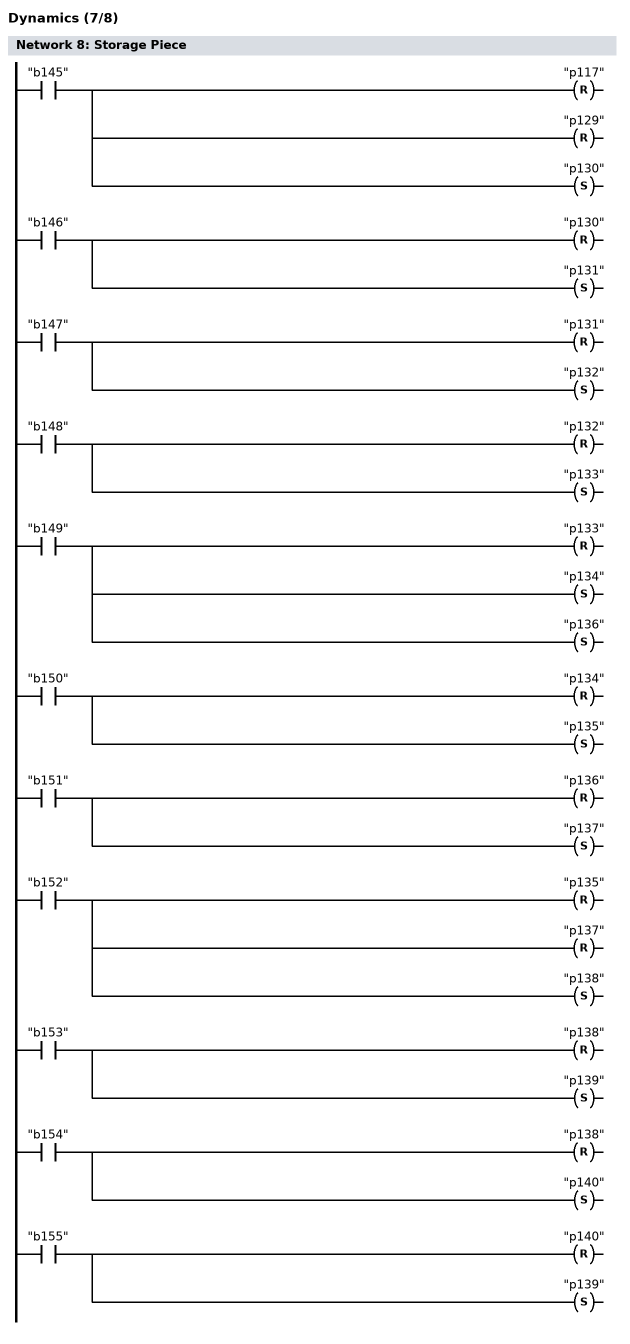
   RUNG wire#powerrail
      Contact( "b145" )
      wire#w1
      R_Coil( "p117" )
   END_RUNG
   RUNG wire#w1
      R_Coil( "p129" )
   END_RUNG
   RUNG wire#w1
      S_Coil( "p130" )
   END_RUNG
   RUNG wire#powerrail
      Contact( "b146" )
      wire#w2
      R_Coil( "p130" )
   END_RUNG
   RUNG wire#w2
      S_Coil( "p131" )
   END_RUNG
   RUNG wire#powerrail
      Contact( "b147" )
      wire#w3
      R_Coil( "p131" )
   END_RUNG
   RUNG wire#w3
      S_Coil( "p132" )
   END_RUNG
   RUNG wire#powerrail
      Contact( "b148" )
      wire#w4
      R_Coil( "p132" )
   END_RUNG
   RUNG wire#w4
      S_Coil( "p133" )
   END_RUNG
   RUNG wire#powerrail
      Contact( "b149" )
      wire#w5
      R_Coil( "p133" )
   END_RUNG
   RUNG wire#w5
      S_Coil( "p134" )
   END_RUNG
   RUNG wire#w5
      S_Coil( "p136" )
   END_RUNG
   RUNG wire#powerrail
      Contact( "b150" )
      wire#w6
      R_Coil( "p134" )
   END_RUNG
   RUNG wire#w6
      S_Coil( "p135" )
   END_RUNG
   RUNG wire#powerrail
      Contact( "b151" )
      wire#w7
      R_Coil( "p136" )
   END_RUNG
   RUNG wire#w7
      S_Coil( "p137" )
   END_RUNG
   RUNG wire#powerrail
      Contact( "b152" )
      wire#w8
      R_Coil( "p135" )
   END_RUNG
   RUNG wire#w8
      R_Coil( "p137" )
   END_RUNG
   RUNG wire#w8
      S_Coil( "p138" )
   END_RUNG
   RUNG wire#powerrail
      Contact( "b153" )
      wire#w9
      R_Coil( "p138" )
   END_RUNG
   RUNG wire#w9
      S_Coil( "p139" )
   END_RUNG
   RUNG wire#powerrail
      Contact( "b154" )
      wire#w10
      R_Coil( "p138" )
   END_RUNG
   RUNG wire#w10
      S_Coil( "p140" )
   END_RUNG
   RUNG wire#powerrail
      Contact( "b155" )
      wire#w11
      R_Coil( "p140" )
   END_RUNG
   RUNG wire#w11
      S_Coil( "p139" )
   END_RUNG
   // the same network as SCL:
   IF "b145" THEN
       "p117" := FALSE;
       "p129" := FALSE;
       "p130" := TRUE;
   END_IF;
   IF "b146" THEN
       "p130" := FALSE;
       "p131" := TRUE;
   END_IF;
   IF "b147" THEN
       "p131" := FALSE;
       "p132" := TRUE;
   END_IF;
   IF "b148" THEN
       "p132" := FALSE;
       "p133" := TRUE;
   END_IF;
   IF "b149" THEN
       "p133" := FALSE;
       "p134" := TRUE;
       "p136" := TRUE;
   END_IF;
   IF "b150" THEN
       "p134" := FALSE;
       "p135" := TRUE;
   END_IF;
   IF "b151" THEN
       "p136" := FALSE;
       "p137" := TRUE;
   END_IF;
   IF "b152" THEN
       "p135" := FALSE;
       "p137" := FALSE;
       "p138" := TRUE;
   END_IF;
   IF "b153" THEN
       "p138" := FALSE;
       "p139" := TRUE;
   END_IF;
   IF "b154" THEN
       "p138" := FALSE;
       "p140" := TRUE;
   END_IF;
   IF "b155" THEN
       "p140" := FALSE;
       "p139" := TRUE;
   END_IF;
END_REGION

REGION Network 9: Arm Stop pt2
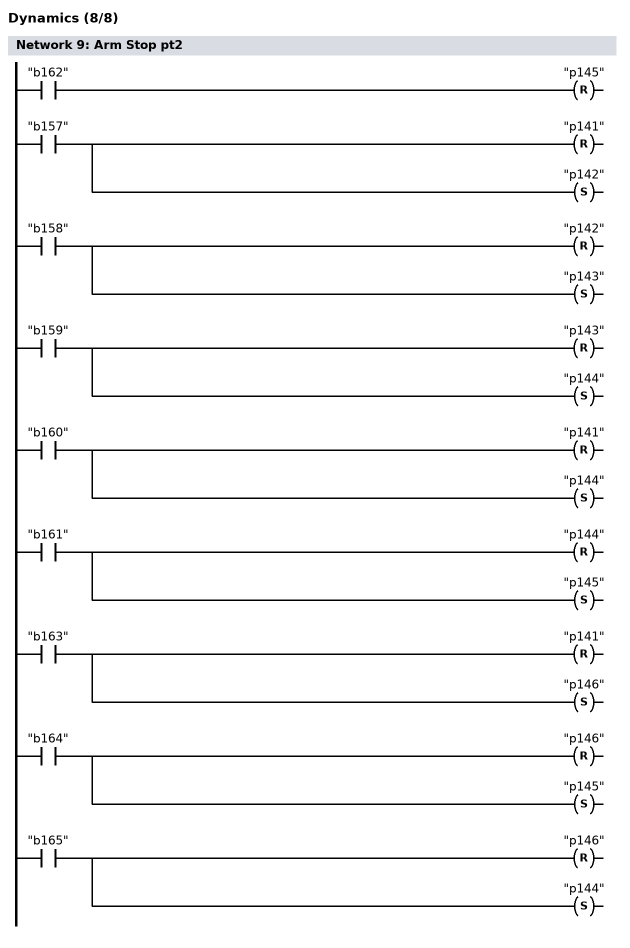
   RUNG wire#powerrail
      Contact( "b162" )
      R_Coil( "p145" )
   END_RUNG
   RUNG wire#powerrail
      Contact( "b157" )
      wire#w1
      R_Coil( "p141" )
   END_RUNG
   RUNG wire#w1
      S_Coil( "p142" )
   END_RUNG
   RUNG wire#powerrail
      Contact( "b158" )
      wire#w2
      R_Coil( "p142" )
   END_RUNG
   RUNG wire#w2
      S_Coil( "p143" )
   END_RUNG
   RUNG wire#powerrail
      Contact( "b159" )
      wire#w3
      R_Coil( "p143" )
   END_RUNG
   RUNG wire#w3
      S_Coil( "p144" )
   END_RUNG
   RUNG wire#powerrail
      Contact( "b160" )
      wire#w4
      R_Coil( "p141" )
   END_RUNG
   RUNG wire#w4
      S_Coil( "p144" )
   END_RUNG
   RUNG wire#powerrail
      Contact( "b161" )
      wire#w5
      R_Coil( "p144" )
   END_RUNG
   RUNG wire#w5
      S_Coil( "p145" )
   END_RUNG
   RUNG wire#powerrail
      Contact( "b163" )
      wire#w6
      R_Coil( "p141" )
   END_RUNG
   RUNG wire#w6
      S_Coil( "p146" )
   END_RUNG
   RUNG wire#powerrail
      Contact( "b164" )
      wire#w7
      R_Coil( "p146" )
   END_RUNG
   RUNG wire#w7
      S_Coil( "p145" )
   END_RUNG
   RUNG wire#powerrail
      Contact( "b165" )
      wire#w8
      R_Coil( "p146" )
   END_RUNG
   RUNG wire#w8
      S_Coil( "p144" )
   END_RUNG
   // the same network as SCL:
   IF "b162" THEN "p145" := FALSE; END_IF;
   IF "b157" THEN
       "p141" := FALSE;
       "p142" := TRUE;
   END_IF;
   IF "b158" THEN
       "p142" := FALSE;
       "p143" := TRUE;
   END_IF;
   IF "b159" THEN
       "p143" := FALSE;
       "p144" := TRUE;
   END_IF;
   IF "b160" THEN
       "p141" := FALSE;
       "p144" := TRUE;
   END_IF;
   IF "b161" THEN
       "p144" := FALSE;
       "p145" := TRUE;
   END_IF;
   IF "b163" THEN
       "p141" := FALSE;
       "p146" := TRUE;
   END_IF;
   IF "b164" THEN
       "p146" := FALSE;
       "p145" := TRUE;
   END_IF;
   IF "b165" THEN
       "p146" := FALSE;
       "p144" := TRUE;
   END_IF;
END_REGION

REGION Network 10 (SCL): Arm Stop pt1
   IF "b156_StopAll" THEN
       // Statement section IF
       "p141" := 1;
       "p14" := 0;
       "p15" := 0;
       "p16" := 0;
       "p17" := 0;
       "p18" := 0;
       "p19" := 0;
       "p20" := 0;
       "p21" := 0;
       "p22" := 0;
       "p23" := 0;
       "p24" := 0;
       "p25" := 0;
       "p26" := 0;
       "p74" := 0;
       "p75" := 0;
       "p76" := 0;
       "p77" := 0;
       "p78" := 0;
       "p79" := 0;
       "p80" := 0;
       "p81" := 0;
       "p82" := 0;
       "p83" := 0;
       "p84" := 0;
       "p85" := 0;
       "p86" := 0;
       "p87" := 0;
       "p88" := 0;
       "p89" := 0;
       "p90" := 0;
       "p91" := 0;
       "p92" := 0;
       "p93" := 0;
       "p94" := 0;
       "p95" := 0;
       "p96" := 0;
       "p97" := 0;
       "p98" := 0;
       "p99" := 0;
       "p100" := 0;
       "p101" := 0;
       "p102" := 0;
       "p103" := 0;
       "p104" := 0;
       "p105" := 0;
       "p106" := 0;
       "p107" := 0;
       "p108" := 0;
       "p109" := 0;
       "p110" := 0;
       "p111" := 0;
       "p112" := 0;
       "p113" := 0;
       "p114" := 0;
       "p115" := 0;
       "p116" := 0;
       "p117" := 0;
       "p118" := 0;
       "p119" := 0;
       "p120" := 0;
       "p121" := 0;
       "p122" := 0;
       "p123" := 0;
       "p124" := 0;
       "p125" := 0;
       "p126" := 0;
       "p127" := 0;
       "p128" := 0;
       "p129" := 0;
       "p130" := 0;
       "p131" := 0;
       "p132" := 0;
       "p133" := 0;
       "p134" := 0;
       "p135" := 0;
       "p136" := 0;
       "p137" := 0;
       "p138" := 0;
       "p139" := 0;
       "p13" := 0;
       "p140" := 0;
       "p145" := 0;
       "p142" := 0;
       "p143" := 0;
       "p144" := 0;
       "p146" := 0;
   END_IF;
END_REGION
END_FUNCTION

FUNCTION "Initialization" : Void   // FC4, LAD
{ S7_Optimized_Access := 'TRUE' }
VERSION : 0.1
BEGIN
END_FUNCTION

FUNCTION "Actions" : Void   // FC5, LAD
{ S7_Optimized_Access := 'TRUE' }
VERSION : 0.1
BEGIN

REGION Network 1: HalfPieceCounter
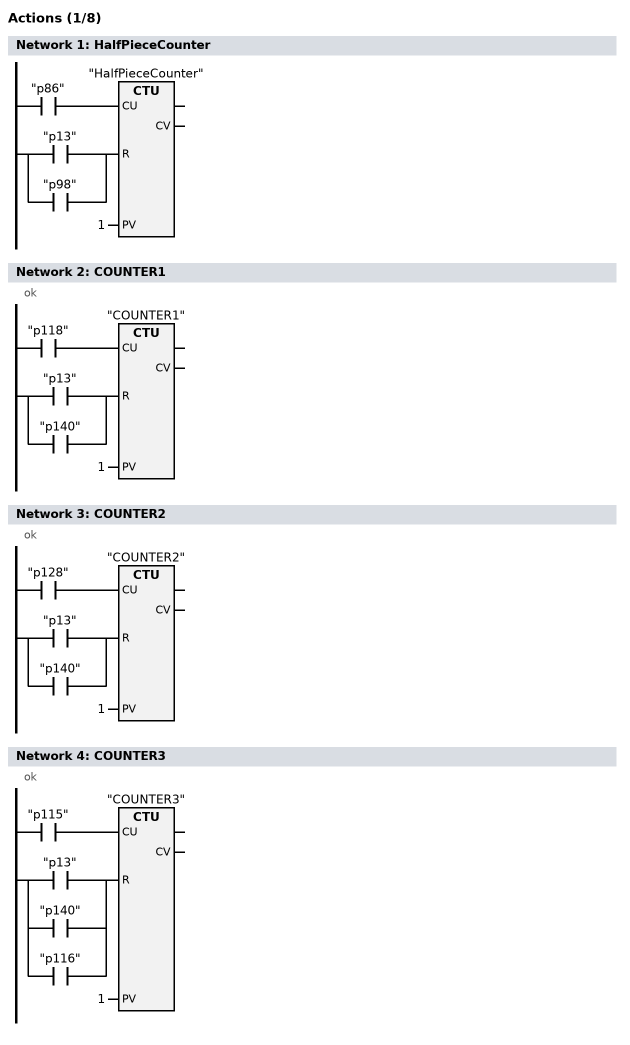
   "HalfPieceCounter".CTU(CU := "p86", R := "p13" OR "p98", PV := 1);
END_REGION

REGION Network 2: COUNTER1
   // ok
   "COUNTER1".CTU(CU := "p118", R := "p13" OR "p140", PV := 1);
END_REGION

REGION Network 3: COUNTER2
   // ok
   "COUNTER2".CTU(CU := "p128", R := "p13" OR "p140", PV := 1);
END_REGION

REGION Network 4: COUNTER3
   // ok
   "COUNTER3".CTU(CU := "p115", R := "p13" OR "p140" OR "p116", PV := 1);
END_REGION

REGION Network 5: COUNTER4
   // ok
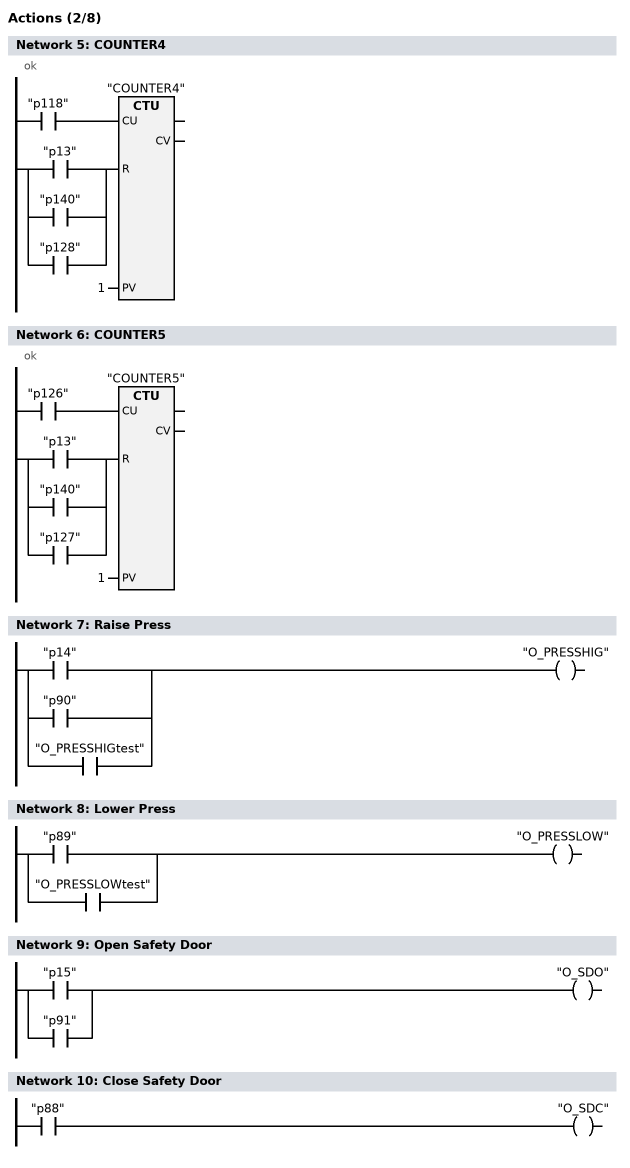
   "COUNTER4".CTU(CU := "p118", R := "p13" OR "p140" OR "p128", PV := 1);
END_REGION

REGION Network 6: COUNTER5
   // ok
   "COUNTER5".CTU(CU := "p126", R := "p13" OR "p140" OR "p127", PV := 1);
END_REGION

REGION Network 7: Raise Press
   RUNG wire#powerrail
      Contact( "p14" )
      wire#w1
      Coil( "O_PRESSHIG" )
   END_RUNG
   RUNG wire#powerrail
      Contact( "p90" )
   END_RUNG wire#w1
   RUNG wire#powerrail
      Contact( "O_PRESSHIGtest" )
   END_RUNG wire#w1
   // the same network as SCL:
   "O_PRESSHIG" := "p14" OR "p90" OR "O_PRESSHIGtest";
END_REGION

REGION Network 8: Lower Press
   RUNG wire#powerrail
      Contact( "p89" )
      wire#w1
      Coil( "O_PRESSLOW" )
   END_RUNG
   RUNG wire#powerrail
      Contact( "O_PRESSLOWtest" )
   END_RUNG wire#w1
   // the same network as SCL:
   "O_PRESSLOW" := "p89" OR "O_PRESSLOWtest";
END_REGION

REGION Network 9: Open Safety Door
   RUNG wire#powerrail
      Contact( "p15" )
      wire#w1
      Coil( "O_SDO" )
   END_RUNG
   RUNG wire#powerrail
      Contact( "p91" )
   END_RUNG wire#w1
   // the same network as SCL:
   "O_SDO" := "p15" OR "p91";
END_REGION

REGION Network 10: Close Safety Door
   RUNG wire#powerrail
      Contact( "p88" )
      Coil( "O_SDC" )
   END_RUNG
   // the same network as SCL:
   "O_SDC" := "p88";
END_REGION

REGION Network 11: Extend Assembly Unit Holder
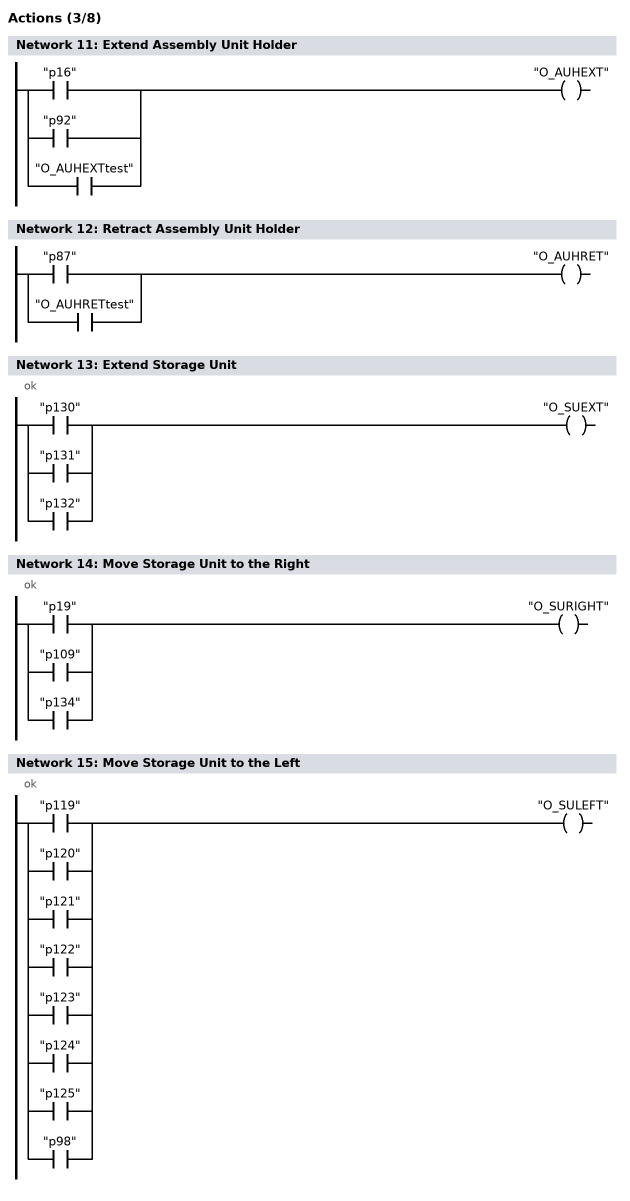
   RUNG wire#powerrail
      Contact( "p16" )
      wire#w1
      Coil( "O_AUHEXT" )
   END_RUNG
   RUNG wire#powerrail
      Contact( "p92" )
   END_RUNG wire#w1
   RUNG wire#powerrail
      Contact( "O_AUHEXTtest" )
   END_RUNG wire#w1
   // the same network as SCL:
   "O_AUHEXT" := "p16" OR "p92" OR "O_AUHEXTtest";
END_REGION

REGION Network 12: Retract Assembly Unit Holder
   RUNG wire#powerrail
      Contact( "p87" )
      wire#w1
      Coil( "O_AUHRET" )
   END_RUNG
   RUNG wire#powerrail
      Contact( "O_AUHRETtest" )
   END_RUNG wire#w1
   // the same network as SCL:
   "O_AUHRET" := "p87" OR "O_AUHRETtest";
END_REGION

REGION Network 13: Extend Storage Unit
   // ok
   RUNG wire#powerrail
      Contact( "p130" )
      wire#w1
      Coil( "O_SUEXT" )
   END_RUNG
   RUNG wire#powerrail
      Contact( "p131" )
   END_RUNG wire#w1
   RUNG wire#powerrail
      Contact( "p132" )
   END_RUNG wire#w1
   // the same network as SCL:
   "O_SUEXT" := "p130" OR "p131" OR "p132";
END_REGION

REGION Network 14: Move Storage Unit to the Right
   // ok
   RUNG wire#powerrail
      Contact( "p19" )
      wire#w1
      Coil( "O_SURIGHT" )
   END_RUNG
   RUNG wire#powerrail
      Contact( "p109" )
   END_RUNG wire#w1
   RUNG wire#powerrail
      Contact( "p134" )
   END_RUNG wire#w1
   // the same network as SCL:
   "O_SURIGHT" := "p19" OR "p109" OR "p134";
END_REGION

REGION Network 15: Move Storage Unit to the Left
   // ok
   RUNG wire#powerrail
      Contact( "p119" )
      wire#w1
      Coil( "O_SULEFT" )
   END_RUNG
   RUNG wire#powerrail
      Contact( "p120" )
   END_RUNG wire#w1
   RUNG wire#powerrail
      Contact( "p121" )
   END_RUNG wire#w1
   RUNG wire#powerrail
      Contact( "p122" )
   END_RUNG wire#w1
   RUNG wire#powerrail
      Contact( "p123" )
   END_RUNG wire#w1
   RUNG wire#powerrail
      Contact( "p124" )
   END_RUNG wire#w1
   RUNG wire#powerrail
      Contact( "p125" )
   END_RUNG wire#w1
   RUNG wire#powerrail
      Contact( "p98" )
   END_RUNG wire#w1
   // the same network as SCL:
   "O_SULEFT" := "p119" OR "p120" OR "p121" OR "p122" OR "p123" OR "p124" OR "p125" OR "p98";
END_REGION

REGION Network 16: Move Storage Unit Downwards
   // ok
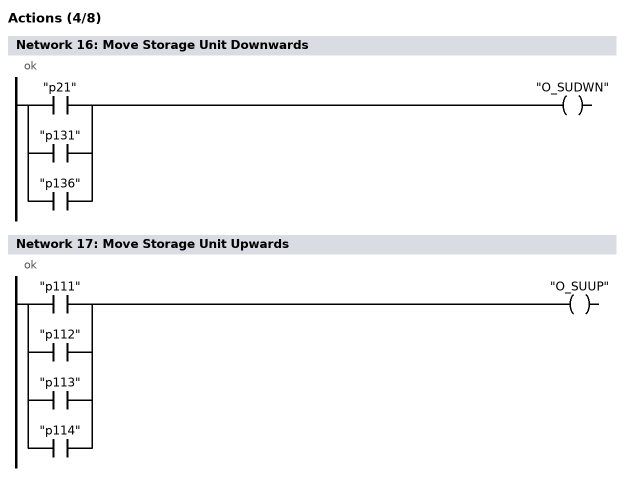
   RUNG wire#powerrail
      Contact( "p21" )
      wire#w1
      Coil( "O_SUDWN" )
   END_RUNG
   RUNG wire#powerrail
      Contact( "p131" )
   END_RUNG wire#w1
   RUNG wire#powerrail
      Contact( "p136" )
   END_RUNG wire#w1
   // the same network as SCL:
   "O_SUDWN" := "p21" OR "p131" OR "p136";
END_REGION

REGION Network 17: Move Storage Unit Upwards
   // ok
   RUNG wire#powerrail
      Contact( "p111" )
      wire#w1
      Coil( "O_SUUP" )
   END_RUNG
   RUNG wire#powerrail
      Contact( "p112" )
   END_RUNG wire#w1
   RUNG wire#powerrail
      Contact( "p113" )
   END_RUNG wire#w1
   RUNG wire#powerrail
      Contact( "p114" )
   END_RUNG wire#w1
   // the same network as SCL:
   "O_SUUP" := "p111" OR "p112" OR "p113" OR "p114";
END_REGION

REGION Network 18: Raise Arm
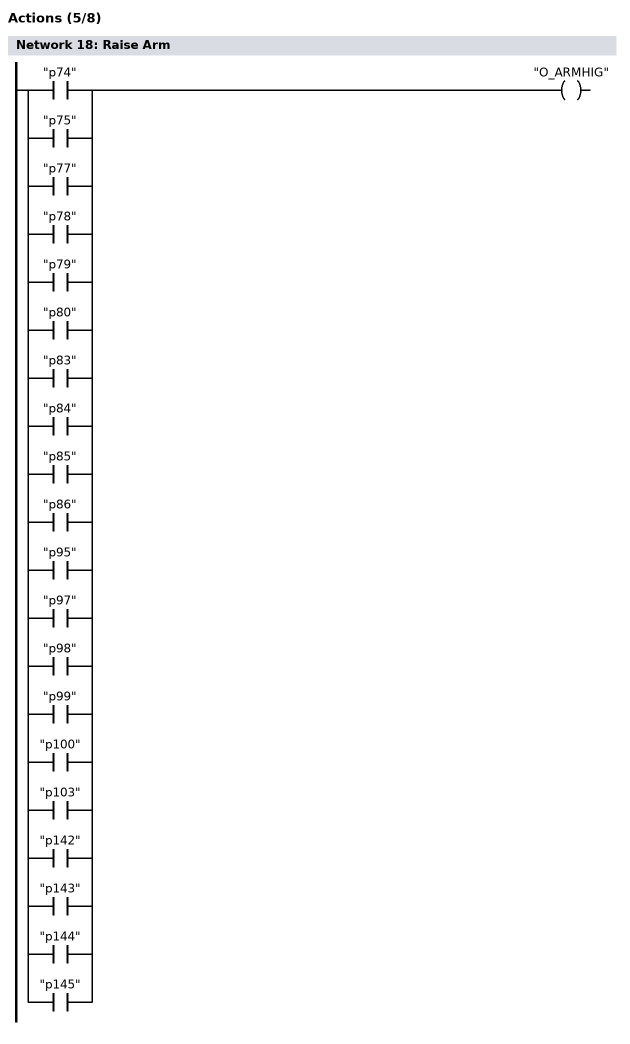
   RUNG wire#powerrail
      Contact( "p74" )
      wire#w1
      Coil( "O_ARMHIG" )
   END_RUNG
   RUNG wire#powerrail
      Contact( "p75" )
   END_RUNG wire#w1
   RUNG wire#powerrail
      Contact( "p77" )
   END_RUNG wire#w1
   RUNG wire#powerrail
      Contact( "p78" )
   END_RUNG wire#w1
   RUNG wire#powerrail
      Contact( "p79" )
   END_RUNG wire#w1
   RUNG wire#powerrail
      Contact( "p80" )
   END_RUNG wire#w1
   RUNG wire#powerrail
      Contact( "p83" )
   END_RUNG wire#w1
   RUNG wire#powerrail
      Contact( "p84" )
   END_RUNG wire#w1
   RUNG wire#powerrail
      Contact( "p85" )
   END_RUNG wire#w1
   RUNG wire#powerrail
      Contact( "p86" )
   END_RUNG wire#w1
   RUNG wire#powerrail
      Contact( "p95" )
   END_RUNG wire#w1
   RUNG wire#powerrail
      Contact( "p97" )
   END_RUNG wire#w1
   RUNG wire#powerrail
      Contact( "p98" )
   END_RUNG wire#w1
   RUNG wire#powerrail
      Contact( "p99" )
   END_RUNG wire#w1
   RUNG wire#powerrail
      Contact( "p100" )
   END_RUNG wire#w1
   RUNG wire#powerrail
      Contact( "p103" )
   END_RUNG wire#w1
   RUNG wire#powerrail
      Contact( "p142" )
   END_RUNG wire#w1
   RUNG wire#powerrail
      Contact( "p143" )
   END_RUNG wire#w1
   RUNG wire#powerrail
      Contact( "p144" )
   END_RUNG wire#w1
   RUNG wire#powerrail
      Contact( "p145" )
   END_RUNG wire#w1
   // the same network as SCL:
   "O_ARMHIG" := "p74" OR "p75" OR "p77" OR "p78" OR "p79" OR "p80" OR "p83" OR "p84" OR "p85" OR "p86" OR "p95" OR "p97" OR "p98" OR "p99" OR "p100" OR "p103" OR "p142" OR "p143" OR "p144" OR "p145";
END_REGION

REGION Network 19: Extend Arm
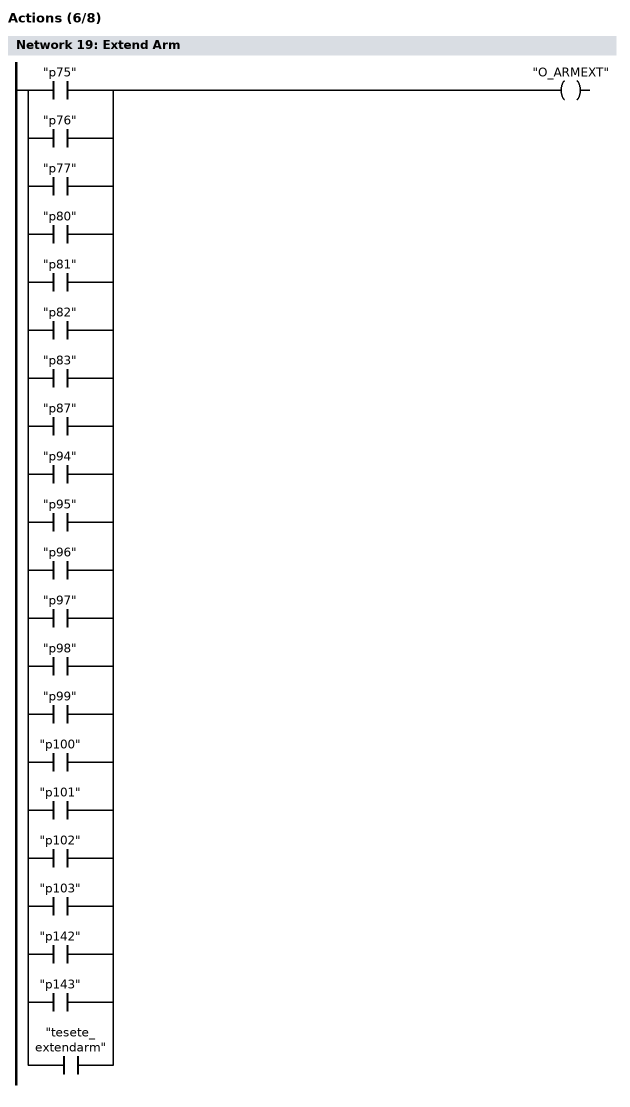
   RUNG wire#powerrail
      Contact( "p75" )
      wire#w1
      Coil( "O_ARMEXT" )
   END_RUNG
   RUNG wire#powerrail
      Contact( "p76" )
   END_RUNG wire#w1
   RUNG wire#powerrail
      Contact( "p77" )
   END_RUNG wire#w1
   RUNG wire#powerrail
      Contact( "p80" )
   END_RUNG wire#w1
   RUNG wire#powerrail
      Contact( "p81" )
   END_RUNG wire#w1
   RUNG wire#powerrail
      Contact( "p82" )
   END_RUNG wire#w1
   RUNG wire#powerrail
      Contact( "p83" )
   END_RUNG wire#w1
   RUNG wire#powerrail
      Contact( "p87" )
   END_RUNG wire#w1
   RUNG wire#powerrail
      Contact( "p94" )
   END_RUNG wire#w1
   RUNG wire#powerrail
      Contact( "p95" )
   END_RUNG wire#w1
   RUNG wire#powerrail
      Contact( "p96" )
   END_RUNG wire#w1
   RUNG wire#powerrail
      Contact( "p97" )
   END_RUNG wire#w1
   RUNG wire#powerrail
      Contact( "p98" )
   END_RUNG wire#w1
   RUNG wire#powerrail
      Contact( "p99" )
   END_RUNG wire#w1
   RUNG wire#powerrail
      Contact( "p100" )
   END_RUNG wire#w1
   RUNG wire#powerrail
      Contact( "p101" )
   END_RUNG wire#w1
   RUNG wire#powerrail
      Contact( "p102" )
   END_RUNG wire#w1
   RUNG wire#powerrail
      Contact( "p103" )
   END_RUNG wire#w1
   RUNG wire#powerrail
      Contact( "p142" )
   END_RUNG wire#w1
   RUNG wire#powerrail
      Contact( "p143" )
   END_RUNG wire#w1
   RUNG wire#powerrail
      Contact( "tesete_extendarm" )
   END_RUNG wire#w1
   // the same network as SCL:
   "O_ARMEXT" := "p75" OR "p76" OR "p77" OR "p80" OR "p81" OR "p82" OR "p83" OR "p87" OR "p94" OR "p95" OR "p96" OR "p97" OR "p98" OR "p99" OR "p100" OR "p101" OR "p102" OR "p103" OR "p142" OR "p143" OR "tesete_extendarm";
END_REGION

REGION Network 20: Turn Vacuum Gripper ON
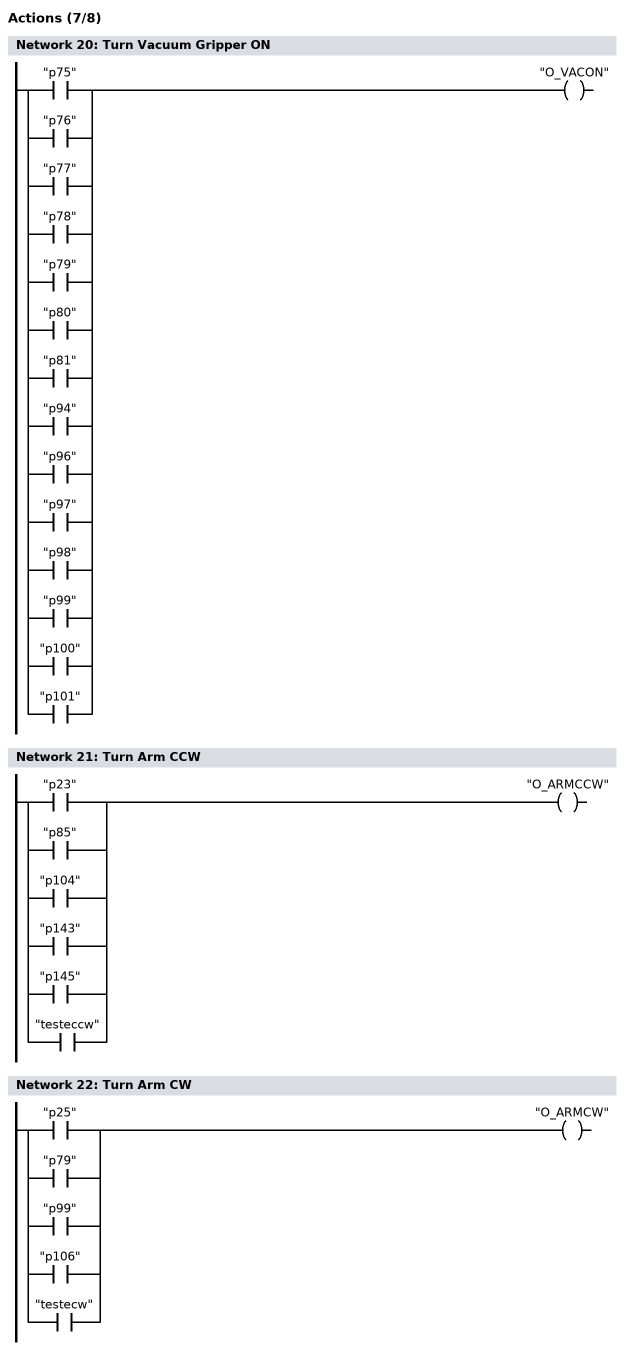
   RUNG wire#powerrail
      Contact( "p75" )
      wire#w1
      Coil( "O_VACON" )
   END_RUNG
   RUNG wire#powerrail
      Contact( "p76" )
   END_RUNG wire#w1
   RUNG wire#powerrail
      Contact( "p77" )
   END_RUNG wire#w1
   RUNG wire#powerrail
      Contact( "p78" )
   END_RUNG wire#w1
   RUNG wire#powerrail
      Contact( "p79" )
   END_RUNG wire#w1
   RUNG wire#powerrail
      Contact( "p80" )
   END_RUNG wire#w1
   RUNG wire#powerrail
      Contact( "p81" )
   END_RUNG wire#w1
   RUNG wire#powerrail
      Contact( "p94" )
   END_RUNG wire#w1
   RUNG wire#powerrail
      Contact( "p96" )
   END_RUNG wire#w1
   RUNG wire#powerrail
      Contact( "p97" )
   END_RUNG wire#w1
   RUNG wire#powerrail
      Contact( "p98" )
   END_RUNG wire#w1
   RUNG wire#powerrail
      Contact( "p99" )
   END_RUNG wire#w1
   RUNG wire#powerrail
      Contact( "p100" )
   END_RUNG wire#w1
   RUNG wire#powerrail
      Contact( "p101" )
   END_RUNG wire#w1
   // the same network as SCL:
   "O_VACON" := "p75" OR "p76" OR "p77" OR "p78" OR "p79" OR "p80" OR "p81" OR "p94" OR "p96" OR "p97" OR "p98" OR "p99" OR "p100" OR "p101";
END_REGION

REGION Network 21: Turn Arm CCW
   RUNG wire#powerrail
      Contact( "p23" )
      wire#w1
      Coil( "O_ARMCCW" )
   END_RUNG
   RUNG wire#powerrail
      Contact( "p85" )
   END_RUNG wire#w1
   RUNG wire#powerrail
      Contact( "p104" )
   END_RUNG wire#w1
   RUNG wire#powerrail
      Contact( "p143" )
   END_RUNG wire#w1
   RUNG wire#powerrail
      Contact( "p145" )
   END_RUNG wire#w1
   RUNG wire#powerrail
      Contact( "testeccw" )
   END_RUNG wire#w1
   // the same network as SCL:
   "O_ARMCCW" := "p23" OR "p85" OR "p104" OR "p143" OR "p145" OR "testeccw";
END_REGION

REGION Network 22: Turn Arm CW
   RUNG wire#powerrail
      Contact( "p25" )
      wire#w1
      Coil( "O_ARMCW" )
   END_RUNG
   RUNG wire#powerrail
      Contact( "p79" )
   END_RUNG wire#w1
   RUNG wire#powerrail
      Contact( "p99" )
   END_RUNG wire#w1
   RUNG wire#powerrail
      Contact( "p106" )
   END_RUNG wire#w1
   RUNG wire#powerrail
      Contact( "testecw" )
   END_RUNG wire#w1
   // the same network as SCL:
   "O_ARMCW" := "p25" OR "p79" OR "p99" OR "p106" OR "testecw";
END_REGION

REGION Network 23: HSC
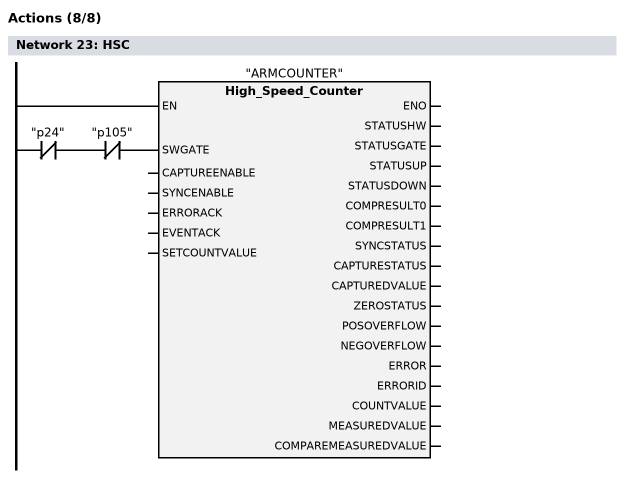
   "ARMCOUNTER"(SwGate := NOT "p24" AND NOT "p105");   // High_Speed_Counter
END_REGION
END_FUNCTION